LIN {X 0,Y 522.499,Z 557.03,A -85,B 0,C 180,E1 4654.238,E2 4654.238} C_VEL
LIN {X 0,Y 522.631,Z 557.03,A -85,B 0,C 180,E1 4659.658,E2 4659.658} C_VEL
LIN {X 0,Y 522.497,Z 557.03,A -85,B 0,C 180,E1 4664.884,E2 4664.884} C_VEL
LIN {X 0,Y 522.702,Z 557.03,A -85,B 0,C 180,E1 4670.012,E2 4670.012} C_VEL
LIN {X 0,Y 522.868,Z 557.03,A -85,B 0,C 180,E1 4675.016,E2 4675.016} C_VEL
LIN {X 0,Y 522.928,Z 557.03,A -85,B 0,C 180,E1 4680,E2 4680} C_VEL
LIN {X 0,Y 522.866,Z 557.03,A -85,B 0,C 180,E1 4684.983,E2 4684.983} C_VEL
LIN {X 0,Y 522.762,Z 557.03,A -85,B 0,C 180,E1 4690.025,E2 4690.025} C_VEL
LIN {X 0,Y 522.691,Z 557.03,A -85,B 0,C 180,E1 4695.11,E2 4695.11} C_VEL
LIN {X 0,Y 522.622,Z 557.03,A -85,B 0,C 180,E1 4700.341,E2 4700.341} C_VEL
LIN {X 0,Y 522.441,Z 557.03,A -85,B 0,C 180,E1 4706.052,E2 4706.052} C_VEL
LIN {X 0,Y 522.368,Z 557.03,A -85,B 0,C 180,E1 4711.445,E2 4711.445} C_VEL
LIN {X 0,Y 522.262,Z 557.03,A -85,B 0,C 180,E1 4717.499,E2 4717.499} C_VEL
LIN {X 0,Y 522.346,Z 557.03,A -85,B 0,C 180,E1 4723.561,E2 4723.561} C_VEL
LIN {X 0,Y 522.43,Z 557.03,A -85,B 0,C 180,E1 4728.89,E2 4728.89} C_VEL
LIN {X 0,Y 522.316,Z 557.03,A -85,B 0,C 180,E1 4734.567,E2 4734.567} C_VEL
LIN {X 0,Y 522.477,Z 557.132,A -85,B 0,C 180,E1 4740.056,E2 4740.056} C_VEL
LIN {X 0,Y 533.026,Z 584.562,A -85,B 0,C 180,E1 4741.253,E2 4741.253} C_VEL
LIN {X 0,Y 531.972,Z 621.412,A -85,B 0,C 180,E1 4742.156,E2 4742.156} C_VEL
LIN {X 0,Y 530.472,Z 657.437,A -85,B 0,C 180,E1 4743.703,E2 4743.703} C_VEL
LIN {X 0,Y 528.574,Z 691.879,A -85,B 0,C 180,E1 4745.909,E2 4745.909} C_VEL
LIN {X 0,Y 526.76,Z 722.651,A -85,B 0,C 180,E1 4748.647,E2 4748.647} C_VEL
LIN {X 0,Y 525.154,Z 749.674,A -85,B 0,C 180,E1 4751.879,E2 4751.879} C_VEL
LIN {X 0,Y 524.132,Z 770.932,A -85,B 0,C 180,E1 4755.312,E2 4755.312} C_VEL
LIN {X 0,Y 523.51,Z 787.531,A -85,B 0,C 180,E1 4758.998,E2 4758.998} C_VEL
LIN {X 0,Y 523.319,Z 798.445,A -85,B 0,C 180,E1 4762.519,E2 4762.519} C_VEL
LIN {X 0,Y 523.187,Z 805.714,A -85,B 0,C 180,E1 4766.682,E2 4766.682} C_VEL
LIN {X 0,Y 523.118,Z 807.495,A -85,B 0,C 180,E1 4770,E2 4770} C_VEL
LIN {X 0,Y 523.197,Z 804.909,A -85,B 0,C 180,E1 4773.94,E2 4773.94} C_VEL
LIN {X 0,Y 523.423,Z 797.131,A -85,B 0,C 180,E1 4777.897,E2 4777.897} C_VEL
LIN {X 0,Y 523.665,Z 784.536,A -85,B 0,C 180,E1 4781.676,E2 4781.676} C_VEL
LIN {X 0,Y 524.44,Z 765.964,A -85,B 0,C 180,E1 4785.488,E2 4785.488} C_VEL
LIN {X 0,Y 525.654,Z 741.391,A -85,B 0,C 180,E1 4789.125,E2 4789.125} C_VEL
LIN {X 0,Y 527.287,Z 712.977,A -85,B 0,C 180,E1 4792.217,E2 4792.217} C_VEL
LIN {X 0,Y 529.245,Z 680.156,A -85,B 0,C 180,E1 4794.845,E2 4794.845} C_VEL
LIN {X 0,Y 530.944,Z 645.809,A -85,B 0,C 180,E1 4796.786,E2 4796.786} C_VEL
LIN {X 0,Y 532.346,Z 608.713,A -85,B 0,C 180,E1 4798.141,E2 4798.141} C_VEL
LIN {X 0,Y 532.591,Z 581.575,A -85,B 0,C 180,E1 4798.739,E2 4798.739} C_VEL
LIN {X 0,Y 522.511,Z 557.03,A -85,B 0,C 180,E1 4799.925,E2 4799.925} C_VEL
LIN {X 0,Y 522.295,Z 557.03,A -85,B 0,C 180,E1 4805.746,E2 4805.746} C_VEL
LIN {X 0,Y 522.316,Z 557.03,A -85,B 0,C 180,E1 4811.813,E2 4811.813} C_VEL
LIN {X 0,Y 522.415,Z 557.03,A -85,B 0,C 180,E1 4818.2,E2 4818.2} C_VEL
LIN {X 0,Y 522.306,Z 557.03,A -85,B 0,C 180,E1 4824.57,E2 4824.57} C_VEL
LIN {X 0,Y 522.381,Z 557.03,A -85,B 0,C 180,E1 4830.483,E2 4830.483} C_VEL
LIN {X 0,Y 522.584,Z 557.03,A -85,B 0,C 180,E1 4836.073,E2 4836.073} C_VEL
LIN {X 0,Y 522.688,Z 557.03,A -85,B 0,C 180,E1 4841.421,E2 4841.421} C_VEL
LIN {X 0,Y 522.818,Z 557.03,A -85,B 0,C 180,E1 4846.606,E2 4846.606} C_VEL
LIN {X 0,Y 522.822,Z 557.03,A -85,B 0,C 180,E1 4851.675,E2 4851.675} C_VEL
LIN {X 0,Y 523.008,Z 557.03,A -85,B 0,C 180,E1 4856.681,E2 4856.681} C_VEL
LIN {X 0,Y 523.061,Z 557.03,A -85,B 0,C 180,E1 4861.659,E2 4861.659} C_VEL
LIN {X 0,Y 522.914,Z 557.03,A -85,B 0,C 180,E1 4866.651,E2 4866.651} C_VEL
LIN {X 0,Y 522.728,Z 557.03,A -85,B 0,C 180,E1 4871.697,E2 4871.697} C_VEL
LIN {X 0,Y 522.567,Z 557.03,A -85,B 0,C 180,E1 4877.037,E2 4877.037} C_VEL
LIN {X 0,Y 522.584,Z 557.03,A -85,B 0,C 180,E1 4882.124,E2 4882.124} C_VEL
LIN {X 0,Y 522.459,Z 557.03,A -85,B 0,C 180,E1 4887.622,E2 4887.622} C_VEL
LIN {X 0,Y 522.344,Z 557.03,A -85,B 0,C 180,E1 4892.52,E2 4892.52} C_VEL
LIN {X 0,Y 519.879,Z 557.03,A -85,B 0,C 180,E1 4893.934,E2 4893.934} C_VEL
LIN {X 0,Y 514.507,Z 557.03,A -85,B 0,C 180,E1 4896.053,E2 4896.053} C_VEL
LIN {X 0,Y 514.405,Z 557.03,A -85,B 0,C 180,E1 4896.298,E2 4896.298} C_VEL
LIN {X 0,Y 514.489,Z 557.03,A -85,B 0,C 180,E1 4902.634,E2 4902.634} C_VEL
LIN {X 0,Y 514.412,Z 557.03,A -85,B 0,C 180,E1 4907.395,E2 4907.395} C_VEL
LIN {X 0,Y 514.417,Z 557.03,A -85,B 0,C 180,E1 4913.939,E2 4913.939} C_VEL
LIN {X 0,Y 514.455,Z 557.03,A -85,B 0,C 180,E1 4914.47,E2 4914.47} C_VEL
LIN {X 0,Y 527.108,Z 583.904,A -85,B 0,C 180,E1 4915.848,E2 4915.848} C_VEL
LIN {X 0,Y 529.672,Z 589.378,A -85,B 0,C 180,E1 4916.123,E2 4916.123} C_VEL
LIN {X 0,Y 528.629,Z 631.367,A -85,B 0,C 180,E1 4916.994,E2 4916.994} C_VEL
LIN {X 0,Y 526.749,Z 669.423,A -85,B 0,C 180,E1 4918.414,E2 4918.414} C_VEL
LIN {X 0,Y 524.486,Z 706.242,A -85,B 0,C 180,E1 4920.481,E2 4920.481} C_VEL
LIN {X 0,Y 521.855,Z 740.903,A -85,B 0,C 180,E1 4923.16,E2 4923.16} C_VEL
LIN {X 0,Y 519.397,Z 773.263,A -85,B 0,C 180,E1 4926.513,E2 4926.513} C_VEL
LIN {X 0,Y 517.458,Z 800.955,A -85,B 0,C 180,E1 4930.338,E2 4930.338} C_VEL
LIN {X 0,Y 516.251,Z 822.301,A -85,B 0,C 180,E1 4934.26,E2 4934.26} C_VEL
LIN {X 0,Y 515.569,Z 837.902,A -85,B 0,C 180,E1 4938.138,E2 4938.138} C_VEL
LIN {X 0,Y 515.355,Z 849.538,A -85,B 0,C 180,E1 4942.403,E2 4942.403} C_VEL
LIN {X 0,Y 515.273,Z 855.897,A -85,B 0,C 180,E1 4946.631,E2 4946.631} C_VEL
LIN {X 0,Y 515.214,Z 857.5,A -85,B 0,C 180,E1 4950,E2 4950} C_VEL
LIN {X 0,Y 515.205,Z 855.898,A -85,B 0,C 180,E1 4953.37,E2 4953.37} C_VEL
LIN {X 0,Y 515.345,Z 849.538,A -85,B 0,C 180,E1 4957.597,E2 4957.597} C_VEL
LIN {X 0,Y 515.631,Z 837.901,A -85,B 0,C 180,E1 4961.862,E2 4961.862} C_VEL
LIN {X 0,Y 516.397,Z 820.237,A -85,B 0,C 180,E1 4966.173,E2 4966.173} C_VEL
LIN {X 0,Y 517.695,Z 798.153,A -85,B 0,C 180,E1 4970.099,E2 4970.099} C_VEL
LIN {X 0,Y 519.59,Z 771.372,A -85,B 0,C 180,E1 4973.702,E2 4973.702} C_VEL
LIN {X 0,Y 521.839,Z 740.896,A -85,B 0,C 180,E1 4976.842,E2 4976.842} C_VEL
LIN {X 0,Y 524.41,Z 706.227,A -85,B 0,C 180,E1 4979.524,E2 4979.524} C_VEL
LIN {X 0,Y 526.744,Z 669.005,A -85,B 0,C 180,E1 4981.607,E2 4981.607} C_VEL
LIN {X 0,Y 528.668,Z 630.098,A -85,B 0,C 180,E1 4983.042,E2 4983.042} C_VEL
LIN {X 0,Y 529.166,Z 588.175,A -85,B 0,C 180,E1 4983.933,E2 4983.933} C_VEL
LIN {X 0,Y 514.456,Z 557.03,A -85,B 0,C 180,E1 4985.532,E2 4985.532} C_VEL
LIN {X 0,Y 514.375,Z 557.03,A -85,B 0,C 180,E1 4990.359,E2 4990.359} C_VEL
LIN {X 0,Y 514.417,Z 557.03,A -85,B 0,C 180,E1 4995.063,E2 4995.063} C_VEL
LIN {X 0,Y 514.496,Z 557.03,A -85,B 0,C 180,E1 4999.918,E2 4999.918} C_VEL
LIN {X 0,Y 514.385,Z 557.03,A -85,B 0,C 180,E1 5005.998,E2 5005.998} C_VEL
LIN {X 0,Y 514.51,Z 557.03,A -85,B 0,C 180,E1 5011.984,E2 5011.984} C_VEL
LIN {X 0,Y 514.641,Z 557.03,A -85,B 0,C 180,E1 5017.516,E2 5017.516} C_VEL
LIN {X 0,Y 514.742,Z 557.03,A -85,B 0,C 180,E1 5022.895,E2 5022.895} C_VEL
LIN {X 0,Y 514.768,Z 557.03,A -85,B 0,C 180,E1 5029.836,E2 5029.836} C_VEL
LIN {X 0,Y 514.968,Z 557.03,A -85,B 0,C 180,E1 5034.94,E2 5034.94} C_VEL
LIN {X 0,Y 515.032,Z 557.03,A -85,B 0,C 180,E1 5040,E2 5040} C_VEL
LIN {X 0,Y 514.96,Z 557.03,A -85,B 0,C 180,E1 5045.06,E2 5045.06} C_VEL
LIN {X 0,Y 514.869,Z 557.03,A -85,B 0,C 180,E1 5050.161,E2 5050.161} C_VEL
LIN {X 0,Y 514.779,Z 557.03,A -85,B 0,C 180,E1 5055.348,E2 5055.348} C_VEL
LIN {X 0,Y 514.686,Z 557.03,A -85,B 0,C 180,E1 5060.669,E2 5060.669} C_VEL
LIN {X 0,Y 514.537,Z 557.03,A -85,B 0,C 180,E1 5066.19,E2 5066.19} C_VEL
LIN {X 0,Y 514.479,Z 557.03,A -85,B 0,C 180,E1 5071.984,E2 5071.984} C_VEL
LIN {X 0,Y 514.339,Z 557.03,A -85,B 0,C 180,E1 5078.179,E2 5078.179} C_VEL
LIN {X 0,Y 514.408,Z 557.03,A -85,B 0,C 180,E1 5084.937,E2 5084.937} C_VEL
LIN {X 0,Y 514.5,Z 557.03,A -85,B 0,C 180,E1 5089.912,E2 5089.912} C_VEL
LIN {X 0,Y 514.382,Z 557.03,A -85,B 0,C 180,E1 5095.995,E2 5095.995} C_VEL
LIN {X 0,Y 514.531,Z 557.515,A -85,B 0,C 180,E1 5099.458,E2 5099.458} C_VEL
LIN {X 0,Y 526.353,Z 586.45,A -85,B 0,C 180,E1 5100.821,E2 5100.821} C_VEL
LIN {X 0,Y 525.106,Z 622.044,A -85,B 0,C 180,E1 5101.74,E2 5101.74} C_VEL
LIN {X 0,Y 523.259,Z 658.762,A -85,B 0,C 180,E1 5103.386,E2 5103.386} C_VEL
LIN {X 0,Y 521.147,Z 693.261,A -85,B 0,C 180,E1 5105.658,E2 5105.658} C_VEL
LIN {X 0,Y 519.142,Z 724.17,A -85,B 0,C 180,E1 5108.48,E2 5108.48} C_VEL
LIN {X 0,Y 517.4,Z 751.061,A -85,B 0,C 180,E1 5111.804,E2 5111.804} C_VEL
LIN {X 0,Y 516.257,Z 773.247,A -85,B 0,C 180,E1 5115.545,E2 5115.545} C_VEL
LIN {X 0,Y 515.614,Z 789.381,A -85,B 0,C 180,E1 5119.344,E2 5119.344} C_VEL
LIN {X 0,Y 515.396,Z 800.367,A -85,B 0,C 180,E1 5123.252,E2 5123.252} C_VEL
LIN {X 0,Y 515.204,Z 806.579,A -85,B 0,C 180,E1 5127.564,E2 5127.564} C_VEL
LIN {X 0,Y 515.283,Z 806.982,A -85,B 0,C 180,E1 5131.683,E2 5131.683} C_VEL
LIN {X 0,Y 515.352,Z 801.871,A -85,B 0,C 180,E1 5135.902,E2 5135.902} C_VEL
LIN {X 0,Y 515.538,Z 792.198,A -85,B 0,C 180,E1 5139.722,E2 5139.722} C_VEL
LIN {X 0,Y 516.197,Z 775.889,A -85,B 0,C 180,E1 5143.839,E2 5143.839} C_VEL
LIN {X 0,Y 517.179,Z 754.854,A -85,B 0,C 180,E1 5147.543,E2 5147.543} C_VEL
LIN {X 0,Y 518.68,Z 729.937,A -85,B 0,C 180,E1 5150.797,E2 5150.797} C_VEL
LIN {X 0,Y 520.75,Z 699.762,A -85,B 0,C 180,E1 5153.735,E2 5153.735} C_VEL
LIN {X 0,Y 522.778,Z 667.008,A -85,B 0,C 180,E1 5156.05,E2 5156.05} C_VEL
LIN {X 0,Y 524.759,Z 631.374,A -85,B 0,C 180,E1 5157.815,E2 5157.815} C_VEL
LIN {X 0,Y 526.101,Z 597.165,A -85,B 0,C 180,E1 5158.874,E2 5158.874} C_VEL
LIN {X 0,Y 525.587,Z 583.161,A -85,B 0,C 180,E1 5159.205,E2 5159.205} C_VEL
LIN {X 0,Y 514.561,Z 557.03,A -85,B 0,C 180,E1 5160.492,E2 5160.492} C_VEL
LIN {X 0,Y 514.377,Z 557.03,A -85,B 0,C 180,E1 5166.064,E2 5166.064} C_VEL
LIN {X 0,Y 514.409,Z 557.03,A -85,B 0,C 180,E1 5172.628,E2 5172.628} C_VEL
LIN {X 0,Y 514.486,Z 557.03,A -85,B 0,C 180,E1 5177.406,E2 5177.406} C_VEL
LIN {X 0,Y 514.433,Z 557.03,A -85,B 0,C 180,E1 5182.622,E2 5182.622} C_VEL
LIN {X 0,Y 514.431,Z 557.03,A -85,B 0,C 180,E1 5188.595,E2 5188.595} C_VEL
LIN {X 0,Y 514.608,Z 557.03,A -85,B 0,C 180,E1 5193.814,E2 5193.814} C_VEL
LIN {X 0,Y 514.718,Z 557.03,A -85,B 0,C 180,E1 5200.267,E2 5200.267} C_VEL
LIN {X 0,Y 514.888,Z 557.03,A -85,B 0,C 180,E1 5206.395,E2 5206.395} C_VEL
LIN {X 0,Y 514.935,Z 557.03,A -85,B 0,C 180,E1 5211.547,E2 5211.547} C_VEL
LIN {X 0,Y 515.096,Z 557.03,A -85,B 0,C 180,E1 5216.63,E2 5216.63} C_VEL
LIN {X 0,Y 515.079,Z 557.03,A -85,B 0,C 180,E1 5221.971,E2 5221.971} C_VEL
LIN {X 0,Y 515.004,Z 557.03,A -85,B 0,C 180,E1 5226.753,E2 5226.753} C_VEL
LIN {X 0,Y 514.797,Z 557.03,A -85,B 0,C 180,E1 5231.88,E2 5231.88} C_VEL
LIN {X 0,Y 514.671,Z 557.03,A -85,B 0,C 180,E1 5237.107,E2 5237.107} C_VEL
LIN {X 0,Y 514.639,Z 557.03,A -85,B 0,C 180,E1 5242.485,E2 5242.485} C_VEL
LIN {X 0,Y 514.501,Z 557.03,A -85,B 0,C 180,E1 5248.087,E2 5248.087} C_VEL
LIN {X 0,Y 514.384,Z 557.03,A -85,B 0,C 180,E1 5254.002,E2 5254.002} C_VEL
LIN {X 0,Y 514.405,Z 557.03,A -85,B 0,C 180,E1 5256.298,E2 5256.298} C_VEL
LIN {X 0,Y 513.119,Z 557.03,A -85,B 0,C 180,E1 5257.261,E2 5257.261} C_VEL
LIN {X 0,Y 506.5,Z 557.03,A -85,B 0,C 180,E1 5259.885,E2 5259.885} C_VEL
LIN {X 0,Y 506.412,Z 557.03,A -85,B 0,C 180,E1 5260.134,E2 5260.134} C_VEL
LIN {X 0,Y 506.444,Z 557.03,A -85,B 0,C 180,E1 5265.844,E2 5265.844} C_VEL
LIN {X 0,Y 506.405,Z 557.03,A -85,B 0,C 180,E1 5271.108,E2 5271.108} C_VEL
LIN {X 0,Y 506.542,Z 557.03,A -85,B 0,C 180,E1 5273.919,E2 5273.919} C_VEL
LIN {X 0,Y 517.256,Z 579.74,A -85,B 0,C 180,E1 5275.038,E2 5275.038} C_VEL
LIN {X 0,Y 523.116,Z 591.895,A -85,B 0,C 180,E1 5275.681,E2 5275.681} C_VEL
LIN {X 0,Y 521.907,Z 633.932,A -85,B 0,C 180,E1 5276.594,E2 5276.594} C_VEL
LIN {X 0,Y 519.721,Z 673.354,A -85,B 0,C 180,E1 5278.136,E2 5278.136} C_VEL
LIN {X 0,Y 517.139,Z 711.434,A -85,B 0,C 180,E1 5280.392,E2 5280.392} C_VEL
LIN {X 0,Y 514.294,Z 745.785,A -85,B 0,C 180,E1 5283.206,E2 5283.206} C_VEL
LIN {X 0,Y 511.637,Z 776.353,A -85,B 0,C 180,E1 5286.535,E2 5286.535} C_VEL
LIN {X 0,Y 509.707,Z 802.295,A -85,B 0,C 180,E1 5290.252,E2 5290.252} C_VEL
LIN {X 0,Y 508.425,Z 822.302,A -85,B 0,C 180,E1 5294.011,E2 5294.011} C_VEL
LIN {X 0,Y 507.684,Z 839.28,A -85,B 0,C 180,E1 5298.387,E2 5298.387} C_VEL
LIN {X 0,Y 507.455,Z 849.538,A -85,B 0,C 180,E1 5302.284,E2 5302.284} C_VEL
LIN {X 0,Y 507.366,Z 855.897,A -85,B 0,C 180,E1 5306.579,E2 5306.579} C_VEL
LIN {X 0,Y 507.327,Z 857.5,A -85,B 0,C 180,E1 5310,E2 5310} C_VEL
LIN {X 0,Y 507.305,Z 855.898,A -85,B 0,C 180,E1 5313.422,E2 5313.422} C_VEL
LIN {X 0,Y 507.454,Z 849.538,A -85,B 0,C 180,E1 5317.716,E2 5317.716} C_VEL
LIN {X 0,Y 507.781,Z 837.9,A -85,B 0,C 180,E1 5322.048,E2 5322.048} C_VEL
LIN {X 0,Y 508.634,Z 820.236,A -85,B 0,C 180,E1 5326.427,E2 5326.427} C_VEL
LIN {X 0,Y 510.039,Z 798.151,A -85,B 0,C 180,E1 5330.414,E2 5330.414} C_VEL
LIN {X 0,Y 512.212,Z 770.604,A -85,B 0,C 180,E1 5334.158,E2 5334.158} C_VEL
LIN {X 0,Y 514.731,Z 739.628,A -85,B 0,C 180,E1 5337.362,E2 5337.362} C_VEL
LIN {X 0,Y 517.404,Z 706.224,A -85,B 0,C 180,E1 5339.965,E2 5339.965} C_VEL
LIN {X 0,Y 519.9,Z 669.735,A -85,B 0,C 180,E1 5342.035,E2 5342.035} C_VEL
LIN {X 0,Y 521.975,Z 631.3,A -85,B 0,C 180,E1 5343.484,E2 5343.484} C_VEL
LIN {X 0,Y 522.476,Z 590.576,A -85,B 0,C 180,E1 5344.388,E2 5344.388} C_VEL
LIN {X 0,Y 506.611,Z 558.216,A -85,B 0,C 180,E1 5346.039,E2 5346.039} C_VEL
LIN {X 0,Y 506.517,Z 557.03,A -85,B 0,C 180,E1 5346.195,E2 5346.195} C_VEL
LIN {X 0,Y 506.401,Z 557.03,A -85,B 0,C 180,E1 5351.634,E2 5351.634} C_VEL
LIN {X 0,Y 506.522,Z 557.03,A -85,B 0,C 180,E1 5358.356,E2 5358.356} C_VEL
LIN {X 0,Y 506.529,Z 557.03,A -85,B 0,C 180,E1 5363.809,E2 5363.809} C_VEL
LIN {X 0,Y 506.539,Z 557.03,A -85,B 0,C 180,E1 5370.091,E2 5370.091} C_VEL
LIN {X 0,Y 506.665,Z 557.03,A -85,B 0,C 180,E1 5375.271,E2 5375.271} C_VEL
LIN {X 0,Y 506.836,Z 557.03,A -85,B 0,C 180,E1 5380.817,E2 5380.817} C_VEL
LIN {X 0,Y 506.653,Z 557.03,A -85,B 0,C 180,E1 5386.169,E2 5386.169} C_VEL
LIN {X 0,Y 506.871,Z 557.03,A -85,B 0,C 180,E1 5391.411,E2 5391.411} C_VEL
LIN {X 0,Y 507.009,Z 557.03,A -85,B 0,C 180,E1 5396.576,E2 5396.576} C_VEL
LIN {X 0,Y 507.066,Z 557.03,A -85,B 0,C 180,E1 5401.711,E2 5401.711} C_VEL
LIN {X 0,Y 506.963,Z 557.03,A -85,B 0,C 180,E1 5406.86,E2 5406.86} C_VEL
LIN {X 0,Y 506.862,Z 557.03,A -85,B 0,C 180,E1 5412.068,E2 5412.068} C_VEL
LIN {X 0,Y 506.814,Z 557.03,A -85,B 0,C 180,E1 5417.38,E2 5417.38} C_VEL
LIN {X 0,Y 506.721,Z 557.03,A -85,B 0,C 180,E1 5422.855,E2 5422.855} C_VEL
LIN {X 0,Y 506.529,Z 557.03,A -85,B 0,C 180,E1 5428.569,E2 5428.569} C_VEL
LIN {X 0,Y 506.481,Z 557.03,A -85,B 0,C 180,E1 5434.606,E2 5434.606} C_VEL
LIN {X 0,Y 506.383,Z 557.03,A -85,B 0,C 180,E1 5441.127,E2 5441.127} C_VEL
LIN {X 0,Y 506.49,Z 557.03,A -85,B 0,C 180,E1 5446.564,E2 5446.564} C_VEL
LIN {X 0,Y 506.512,Z 557.03,A -85,B 0,C 180,E1 5453.285,E2 5453.285} C_VEL
LIN {X 0,Y 506.577,Z 557.238,A -85,B 0,C 180,E1 5458.831,E2 5458.831} C_VEL
LIN {X 0,Y 519.682,Z 587.9,A -85,B 0,C 180,E1 5460.364,E2 5460.364} C_VEL
LIN {X 0,Y 518.316,Z 625.057,A -85,B 0,C 180,E1 5461.369,E2 5461.369} C_VEL
LIN {X 0,Y 516.256,Z 660.583,A -85,B 0,C 180,E1 5463.033,E2 5463.033} C_VEL
LIN {X 0,Y 513.847,Z 693.357,A -85,B 0,C 180,E1 5465.289,E2 5465.289} C_VEL
LIN {X 0,Y 511.587,Z 724.917,A -85,B 0,C 180,E1 5468.228,E2 5468.228} C_VEL
LIN {X 0,Y 509.742,Z 751.097,A -85,B 0,C 180,E1 5471.527,E2 5471.527} C_VEL
LIN {X 0,Y 508.46,Z 773.243,A -85,B 0,C 180,E1 5475.318,E2 5475.318} C_VEL
LIN {X 0,Y 507.749,Z 789.668,A -85,B 0,C 180,E1 5479.259,E2 5479.259} C_VEL
LIN {X 0,Y 507.5,Z 800.365,A -85,B 0,C 180,E1 5483.146,E2 5483.146} C_VEL
LIN {X 0,Y 507.388,Z 805.711,A -85,B 0,C 180,E1 5486.578,E2 5486.578} C_VEL
LIN {X 0,Y 507.331,Z 807.495,A -85,B 0,C 180,E1 5490,E2 5490} C_VEL
LIN {X 0,Y 507.423,Z 804.612,A -85,B 0,C 180,E1 5494.278,E2 5494.278} C_VEL
LIN {X 0,Y 507.627,Z 795.988,A -85,B 0,C 180,E1 5498.576,E2 5498.576} C_VEL
LIN {X 0,Y 508.021,Z 782.805,A -85,B 0,C 180,E1 5502.478,E2 5502.478} C_VEL
LIN {X 0,Y 508.94,Z 763.523,A -85,B 0,C 180,E1 5506.416,E2 5506.416} C_VEL
LIN {X 0,Y 510.525,Z 739.65,A -85,B 0,C 180,E1 5509.941,E2 5509.941} C_VEL
LIN {X 0,Y 512.532,Z 711.195,A -85,B 0,C 180,E1 5513.072,E2 5513.072} C_VEL
LIN {X 0,Y 515.048,Z 677.433,A -85,B 0,C 180,E1 5515.812,E2 5515.812} C_VEL
LIN {X 0,Y 517.295,Z 643.917,A -85,B 0,C 180,E1 5517.746,E2 5517.746} C_VEL
LIN {X 0,Y 519.049,Z 607.178,A -85,B 0,C 180,E1 5519.113,E2 5519.113} C_VEL
LIN {X 0,Y 519.234,Z 586.102,A -85,B 0,C 180,E1 5519.613,E2 5519.613} C_VEL
LIN {X 0,Y 506.604,Z 557.03,A -85,B 0,C 180,E1 5521.131,E2 5521.131} C_VEL
LIN {X 0,Y 506.454,Z 557.03,A -85,B 0,C 180,E1 5526.719,E2 5526.719} C_VEL
LIN {X 0,Y 506.448,Z 557.03,A -85,B 0,C 180,E1 5533.44,E2 5533.44} C_VEL
LIN {X 0,Y 506.49,Z 557.03,A -85,B 0,C 180,E1 5538.883,E2 5538.883} C_VEL
LIN {X 0,Y 506.463,Z 557.03,A -85,B 0,C 180,E1 5545.392,E2 5545.392} C_VEL
LIN {X 0,Y 506.535,Z 557.03,A -85,B 0,C 180,E1 5551.432,E2 5551.432} C_VEL
LIN {X 0,Y 506.739,Z 557.03,A -85,B 0,C 180,E1 5557.146,E2 5557.146} C_VEL
LIN {X 0,Y 506.886,Z 557.03,A -85,B 0,C 180,E1 5562.906,E2 5562.906} C_VEL
LIN {X 0,Y 506.913,Z 557.03,A -85,B 0,C 180,E1 5567.933,E2 5567.933} C_VEL
LIN {X 0,Y 506.962,Z 557.03,A -85,B 0,C 180,E1 5573.14,E2 5573.14} C_VEL
LIN {X 0,Y 507.06,Z 557.03,A -85,B 0,C 180,E1 5578.289,E2 5578.289} C_VEL
LIN {X 0,Y 507.003,Z 557.03,A -85,B 0,C 180,E1 5583.424,E2 5583.424} C_VEL
LIN {X 0,Y 506.89,Z 557.03,A -85,B 0,C 180,E1 5588.589,E2 5588.589} C_VEL
LIN {X 0,Y 506.826,Z 557.03,A -85,B 0,C 180,E1 5593.826,E2 5593.826} C_VEL
LIN {X 0,Y 506.71,Z 557.03,A -85,B 0,C 180,E1 5599.188,E2 5599.188} C_VEL
LIN {X 0,Y 506.672,Z 557.03,A -85,B 0,C 180,E1 5604.729,E2 5604.729} C_VEL
LIN {X 0,Y 506.529,Z 557.03,A -85,B 0,C 180,E1 5610.538,E2 5610.538} C_VEL
LIN {X 0,Y 506.522,Z 557.03,A -85,B 0,C 180,E1 5616.711,E2 5616.711} C_VEL
LIN {X 0,Y 506.412,Z 557.03,A -85,B 0,C 180,E1 5620.134,E2 5620.134} C_VEL
LIN {X 0,Y 503.923,Z 557.03,A -85,B 0,C 180,E1 5621.594,E2 5621.594} C_VEL
LIN {X 0,Y 498.652,Z 557.03,A -85,B 0,C 180,E1 5623.784,E2 5623.784} C_VEL
LIN {X 0,Y 498.565,Z 557.03,A -85,B 0,C 180,E1 5624.037,E2 5624.037} C_VEL
LIN {X 0,Y 498.446,Z 557.03,A -85,B 0,C 180,E1 5630.366,E2 5630.366} C_VEL
LIN {X 0,Y 498.625,Z 557.617,A -85,B 0,C 180,E1 5633.375,E2 5633.375} C_VEL
LIN {X 0,Y 516.486,Z 594.362,A -85,B 0,C 180,E1 5635.22,E2 5635.22} C_VEL
LIN {X 0,Y 515.178,Z 636.741,A -85,B 0,C 180,E1 5636.191,E2 5636.191} C_VEL
LIN {X 0,Y 512.771,Z 676.295,A -85,B 0,C 180,E1 5637.814,E2 5637.814} C_VEL
LIN {X 0,Y 509.993,Z 712.973,A -85,B 0,C 180,E1 5640.058,E2 5640.058} C_VEL
LIN {X 0,Y 506.953,Z 746.935,A -85,B 0,C 180,E1 5642.906,E2 5642.906} C_VEL
LIN {X 0,Y 504.073,Z 777.662,A -85,B 0,C 180,E1 5646.336,E2 5646.336} C_VEL
LIN {X 0,Y 501.933,Z 804.002,A -85,B 0,C 180,E1 5650.229,E2 5650.229} C_VEL
LIN {X 0,Y 500.594,Z 824.261,A -85,B 0,C 180,E1 5654.205,E2 5654.205} C_VEL
LIN {X 0,Y 499.831,Z 839.281,A -85,B 0,C 180,E1 5658.202,E2 5658.202} C_VEL
LIN {X 0,Y 499.57,Z 849.538,A -85,B 0,C 180,E1 5662.162,E2 5662.162} C_VEL
LIN {X 0,Y 499.459,Z 855.897,A -85,B 0,C 180,E1 5666.524,E2 5666.524} C_VEL
LIN {X 0,Y 499.444,Z 857.5,A -85,B 0,C 180,E1 5670,E2 5670} C_VEL
LIN {X 0,Y 499.405,Z 855.898,A -85,B 0,C 180,E1 5673.477,E2 5673.477} C_VEL
LIN {X 0,Y 499.577,Z 849.538,A -85,B 0,C 180,E1 5677.839,E2 5677.839} C_VEL
LIN {X 0,Y 499.944,Z 837.9,A -85,B 0,C 180,E1 5682.239,E2 5682.239} C_VEL
LIN {X 0,Y 500.898,Z 820.234,A -85,B 0,C 180,E1 5686.688,E2 5686.688} C_VEL
LIN {X 0,Y 502.454,Z 797.834,A -85,B 0,C 180,E1 5690.786,E2 5690.786} C_VEL
LIN {X 0,Y 504.802,Z 770.245,A -85,B 0,C 180,E1 5694.58,E2 5694.58} C_VEL
LIN {X 0,Y 507.55,Z 739.625,A -85,B 0,C 180,E1 5697.782,E2 5697.782} C_VEL
LIN {X 0,Y 510.447,Z 706.323,A -85,B 0,C 180,E1 5700.409,E2 5700.409} C_VEL
LIN {X 0,Y 513.153,Z 669.732,A -85,B 0,C 180,E1 5702.507,E2 5702.507} C_VEL
LIN {X 0,Y 515.405,Z 630.577,A -85,B 0,C 180,E1 5703.991,E2 5703.991} C_VEL
LIN {X 0,Y 515.916,Z 593.113,A -85,B 0,C 180,E1 5704.841,E2 5704.841} C_VEL
LIN {X 0,Y 498.583,Z 557.03,A -85,B 0,C 180,E1 5706.683,E2 5706.683} C_VEL
LIN {X 0,Y 498.512,Z 557.03,A -85,B 0,C 180,E1 5713.208,E2 5713.208} C_VEL
LIN {X 0,Y 498.54,Z 557.03,A -85,B 0,C 180,E1 5719.398,E2 5719.398} C_VEL
LIN {X 0,Y 498.587,Z 557.03,A -85,B 0,C 180,E1 5725.076,E2 5725.076} C_VEL
LIN {X 0,Y 498.612,Z 557.03,A -85,B 0,C 180,E1 5731.715,E2 5731.715} C_VEL
LIN {X 0,Y 498.762,Z 557.03,A -85,B 0,C 180,E1 5736.758,E2 5736.758} C_VEL
LIN {X 0,Y 498.889,Z 557.03,A -85,B 0,C 180,E1 5742.334,E2 5742.334} C_VEL
LIN {X 0,Y 498.798,Z 557.03,A -85,B 0,C 180,E1 5747.733,E2 5747.733} C_VEL
LIN {X 0,Y 499.15,Z 557.03,A -85,B 0,C 180,E1 5753.031,E2 5753.031} C_VEL
LIN {X 0,Y 499.404,Z 557.03,A -85,B 0,C 180,E1 5758.262,E2 5758.262} C_VEL
LIN {X 0,Y 499.3,Z 557.03,A -85,B 0,C 180,E1 5763.476,E2 5763.476} C_VEL
LIN {X 0,Y 499.096,Z 557.03,A -85,B 0,C 180,E1 5768.723,E2 5768.723} C_VEL
LIN {X 0,Y 498.969,Z 557.03,A -85,B 0,C 180,E1 5774.047,E2 5774.047} C_VEL
LIN {X 0,Y 498.835,Z 557.03,A -85,B 0,C 180,E1 5779.795,E2 5779.795} C_VEL
LIN {X 0,Y 498.727,Z 557.03,A -85,B 0,C 180,E1 5785.149,E2 5785.149} C_VEL
LIN {X 0,Y 498.566,Z 557.03,A -85,B 0,C 180,E1 5791.754,E2 5791.754} C_VEL
LIN {X 0,Y 498.448,Z 557.03,A -85,B 0,C 180,E1 5797.837,E2 5797.837} C_VEL
LIN {X 0,Y 498.524,Z 557.03,A -85,B 0,C 180,E1 5804.304,E2 5804.304} C_VEL
LIN {X 0,Y 498.531,Z 557.03,A -85,B 0,C 180,E1 5810.373,E2 5810.373} C_VEL
LIN {X 0,Y 498.566,Z 557.03,A -85,B 0,C 180,E1 5816.864,E2 5816.864} C_VEL
LIN {X 0,Y 498.65,Z 557.03,A -85,B 0,C 180,E1 5818.152,E2 5818.152} C_VEL
LIN {X 0,Y 512.972,Z 589.835,A -85,B 0,C 180,E1 5819.894,E2 5819.894} C_VEL
LIN {X 0,Y 511.545,Z 628.105,A -85,B 0,C 180,E1 5820.993,E2 5820.993} C_VEL
LIN {X 0,Y 509.316,Z 662.339,A -85,B 0,C 180,E1 5822.659,E2 5822.659} C_VEL
LIN {X 0,Y 506.728,Z 694.383,A -85,B 0,C 180,E1 5824.918,E2 5824.918} C_VEL
LIN {X 0,Y 504.116,Z 725.151,A -85,B 0,C 180,E1 5827.914,E2 5827.914} C_VEL
LIN {X 0,Y 501.992,Z 752.226,A -85,B 0,C 180,E1 5831.408,E2 5831.408} C_VEL
LIN {X 0,Y 500.726,Z 772.632,A -85,B 0,C 180,E1 5834.961,E2 5834.961} C_VEL
LIN {X 0,Y 499.913,Z 788.129,A -85,B 0,C 180,E1 5838.646,E2 5838.646} C_VEL
LIN {X 0,Y 499.663,Z 798.439,A -85,B 0,C 180,E1 5842.163,E2 5842.163} C_VEL
LIN {X 0,Y 499.499,Z 805.71,A -85,B 0,C 180,E1 5846.524,E2 5846.524} C_VEL
LIN {X 0,Y 499.442,Z 807.495,A -85,B 0,C 180,E1 5850,E2 5850} C_VEL
LIN {X 0,Y 499.542,Z 804.613,A -85,B 0,C 180,E1 5854.345,E2 5854.345} C_VEL
LIN {X 0,Y 499.749,Z 795.99,A -85,B 0,C 180,E1 5858.712,E2 5858.712} C_VEL
LIN {X 0,Y 500.182,Z 782.808,A -85,B 0,C 180,E1 5862.677,E2 5862.677} C_VEL
LIN {X 0,Y 501.213,Z 763.526,A -85,B 0,C 180,E1 5866.677,E2 5866.677} C_VEL
LIN {X 0,Y 502.923,Z 739.656,A -85,B 0,C 180,E1 5870.255,E2 5870.255} C_VEL
LIN {X 0,Y 505.531,Z 708.354,A -85,B 0,C 180,E1 5873.754,E2 5873.754} C_VEL
LIN {X 0,Y 508.176,Z 677.074,A -85,B 0,C 180,E1 5876.307,E2 5876.307} C_VEL
LIN {X 0,Y 510.644,Z 643.292,A -85,B 0,C 180,E1 5878.259,E2 5878.259} C_VEL
LIN {X 0,Y 512.475,Z 607.469,A -85,B 0,C 180,E1 5879.598,E2 5879.598} C_VEL
LIN {X 0,Y 512.746,Z 588.544,A -85,B 0,C 180,E1 5880.058,E2 5880.058} C_VEL
LIN {X 0,Y 498.704,Z 557.03,A -85,B 0,C 180,E1 5881.788,E2 5881.788} C_VEL
LIN {X 0,Y 498.449,Z 557.03,A -85,B 0,C 180,E1 5887.843,E2 5887.843} C_VEL
LIN {X 0,Y 498.551,Z 557.03,A -85,B 0,C 180,E1 5894.305,E2 5894.305} C_VEL
LIN {X 0,Y 498.524,Z 557.03,A -85,B 0,C 180,E1 5900.377,E2 5900.377} C_VEL
LIN {X 0,Y 498.525,Z 557.03,A -85,B 0,C 180,E1 5906.864,E2 5906.864} C_VEL
LIN {X 0,Y 498.665,Z 557.03,A -85,B 0,C 180,E1 5912.91,E2 5912.91} C_VEL
LIN {X 0,Y 498.865,Z 557.03,A -85,B 0,C 180,E1 5918.644,E2 5918.644} C_VEL
LIN {X 0,Y 498.99,Z 557.03,A -85,B 0,C 180,E1 5924.154,E2 5924.154} C_VEL
LIN {X 0,Y 499.067,Z 557.03,A -85,B 0,C 180,E1 5929.513,E2 5929.513} C_VEL
LIN {X 0,Y 499.149,Z 557.03,A -85,B 0,C 180,E1 5934.78,E2 5934.78} C_VEL
LIN {X 0,Y 499.277,Z 557.03,A -85,B 0,C 180,E1 5940,E2 5940} C_VEL
LIN {X 0,Y 499.166,Z 557.03,A -85,B 0,C 180,E1 5945.221,E2 5945.221} C_VEL
LIN {X 0,Y 499.013,Z 557.03,A -85,B 0,C 180,E1 5950.488,E2 5950.488} C_VEL
LIN {X 0,Y 498.87,Z 557.03,A -85,B 0,C 180,E1 5955.851,E2 5955.851} C_VEL
LIN {X 0,Y 498.799,Z 557.03,A -85,B 0,C 180,E1 5961.36,E2 5961.36} C_VEL
LIN {X 0,Y 498.652,Z 557.03,A -85,B 0,C 180,E1 5967.092,E2 5967.092} C_VEL
LIN {X 0,Y 498.538,Z 557.03,A -85,B 0,C 180,E1 5973.136,E2 5973.136} C_VEL
LIN {X 0,Y 498.537,Z 557.03,A -85,B 0,C 180,E1 5979.623,E2 5979.623} C_VEL
LIN {X 0,Y 498.565,Z 557.03,A -85,B 0,C 180,E1 5984.037,E2 5984.037} C_VEL
LIN {X 0,Y 496.1,Z 557.03,A -85,B 0,C 180,E1 5985.511,E2 5985.511} C_VEL
LIN {X 0,Y 490.589,Z 557.03,A -85,B 0,C 180,E1 5987.977,E2 5987.977} C_VEL
LIN {X 0,Y 490.617,Z 557.03,A -85,B 0,C 180,E1 5992.765,E2 5992.765} C_VEL
LIN {X 0,Y 509.78,Z 598.268,A -85,B 0,C 180,E1 5994.835,E2 5994.835} C_VEL
LIN {X 0,Y 508.329,Z 638.786,A -85,B 0,C 180,E1 5995.79,E2 5995.79} C_VEL
LIN {X 0,Y 506.046,Z 675.877,A -85,B 0,C 180,E1 5997.309,E2 5997.309} C_VEL
LIN {X 0,Y 503.027,Z 712.969,A -85,B 0,C 180,E1 5999.6,E2 5999.6} C_VEL
LIN {X 0,Y 499.691,Z 747.167,A -85,B 0,C 180,E1 6002.504,E2 6002.504} C_VEL
LIN {X 0,Y 496.638,Z 777.704,A -85,B 0,C 180,E1 6005.966,E2 6005.966} C_VEL
LIN {X 0,Y 494.276,Z 804.226,A -85,B 0,C 180,E1 6009.95,E2 6009.95} C_VEL
LIN {X 0,Y 492.797,Z 824.26,A -85,B 0,C 180,E1 6013.948,E2 6013.948} C_VEL
LIN {X 0,Y 491.971,Z 839.281,A -85,B 0,C 180,E1 6018.011,E2 6018.011} C_VEL
LIN {X 0,Y 491.678,Z 849.538,A -85,B 0,C 180,E1 6022.035,E2 6022.035} C_VEL
LIN {X 0,Y 491.553,Z 855.897,A -85,B 0,C 180,E1 6026.469,E2 6026.469} C_VEL
LIN {X 0,Y 491.544,Z 857.5,A -85,B 0,C 180,E1 6030,E2 6030} C_VEL
LIN {X 0,Y 491.504,Z 855.899,A -85,B 0,C 180,E1 6033.532,E2 6033.532} C_VEL
LIN {X 0,Y 491.69,Z 849.538,A -85,B 0,C 180,E1 6037.965,E2 6037.965} C_VEL
LIN {X 0,Y 492.113,Z 837.899,A -85,B 0,C 180,E1 6042.437,E2 6042.437} C_VEL
LIN {X 0,Y 493.132,Z 820.233,A -85,B 0,C 180,E1 6046.959,E2 6046.959} C_VEL
LIN {X 0,Y 494.845,Z 797.833,A -85,B 0,C 180,E1 6051.121,E2 6051.121} C_VEL
LIN {X 0,Y 497.296,Z 771.445,A -85,B 0,C 180,E1 6054.826,E2 6054.826} C_VEL
LIN {X 0,Y 500.342,Z 740.256,A -85,B 0,C 180,E1 6058.156,E2 6058.156} C_VEL
LIN {X 0,Y 503.53,Z 706.32,A -85,B 0,C 180,E1 6060.872,E2 6060.872} C_VEL
LIN {X 0,Y 506.456,Z 669.495,A -85,B 0,C 180,E1 6063.004,E2 6063.004} C_VEL
LIN {X 0,Y 508.642,Z 631.11,A -85,B 0,C 180,E1 6064.442,E2 6064.442} C_VEL
LIN {X 0,Y 509.102,Z 595.771,A -85,B 0,C 180,E1 6065.254,E2 6065.254} C_VEL
LIN {X 0,Y 490.609,Z 557.03,A -85,B 0,C 180,E1 6067.287,E2 6067.287} C_VEL
LIN {X 0,Y 490.571,Z 557.03,A -85,B 0,C 180,E1 6072.765,E2 6072.765} C_VEL
LIN {X 0,Y 490.691,Z 557.03,A -85,B 0,C 180,E1 6077.777,E2 6077.777} C_VEL
LIN {X 0,Y 490.593,Z 557.03,A -85,B 0,C 180,E1 6084.103,E2 6084.103} C_VEL
LIN {X 0,Y 490.633,Z 557.03,A -85,B 0,C 180,E1 6090.415,E2 6090.415} C_VEL
LIN {X 0,Y 490.834,Z 557.03,A -85,B 0,C 180,E1 6096.36,E2 6096.36} C_VEL
LIN {X 0,Y 490.972,Z 557.03,A -85,B 0,C 180,E1 6102.039,E2 6102.039} C_VEL
LIN {X 0,Y 490.888,Z 557.03,A -85,B 0,C 180,E1 6107.532,E2 6107.532} C_VEL
LIN {X 0,Y 491.223,Z 557.03,A -85,B 0,C 180,E1 6112.918,E2 6112.918} C_VEL
LIN {X 0,Y 491.492,Z 557.03,A -85,B 0,C 180,E1 6118.235,E2 6118.235} C_VEL
LIN {X 0,Y 491.387,Z 557.03,A -85,B 0,C 180,E1 6123.532,E2 6123.532} C_VEL
LIN {X 0,Y 491.113,Z 557.03,A -85,B 0,C 180,E1 6129.414,E2 6129.414} C_VEL
LIN {X 0,Y 491.036,Z 557.03,A -85,B 0,C 180,E1 6134.279,E2 6134.279} C_VEL
LIN {X 0,Y 490.931,Z 557.03,A -85,B 0,C 180,E1 6139.829,E2 6139.829} C_VEL
LIN {X 0,Y 490.755,Z 557.03,A -85,B 0,C 180,E1 6145.587,E2 6145.587} C_VEL
LIN {X 0,Y 490.687,Z 557.03,A -85,B 0,C 180,E1 6151.635,E2 6151.635} C_VEL
LIN {X 0,Y 490.518,Z 557.03,A -85,B 0,C 180,E1 6158.118,E2 6158.118} C_VEL
LIN {X 0,Y 490.614,Z 557.03,A -85,B 0,C 180,E1 6164.782,E2 6164.782} C_VEL
LIN {X 0,Y 490.617,Z 557.03,A -85,B 0,C 180,E1 6170.484,E2 6170.484} C_VEL
LIN {X 0,Y 490.619,Z 557.03,A -85,B 0,C 180,E1 6176.424,E2 6176.424} C_VEL
LIN {X 0,Y 490.732,Z 557.79,A -85,B 0,C 180,E1 6177.518,E2 6177.518} C_VEL
LIN {X 0,Y 506.489,Z 592.242,A -85,B 0,C 180,E1 6179.435,E2 6179.435} C_VEL
LIN {X 0,Y 504.86,Z 629.676,A -85,B 0,C 180,E1 6180.551,E2 6180.551} C_VEL
LIN {X 0,Y 502.435,Z 664.21,A -85,B 0,C 180,E1 6182.277,E2 6182.277} C_VEL
LIN {X 0,Y 499.641,Z 695.659,A -85,B 0,C 180,E1 6184.553,E2 6184.553} C_VEL
LIN {X 0,Y 496.783,Z 726.33,A -85,B 0,C 180,E1 6187.606,E2 6187.606} C_VEL
LIN {X 0,Y 494.276,Z 753.025,A -85,B 0,C 180,E1 6191.232,E2 6191.232} C_VEL
LIN {X 0,Y 492.835,Z 774.861,A -85,B 0,C 180,E1 6195.182,E2 6195.182} C_VEL
LIN {X 0,Y 491.962,Z 791.132,A -85,B 0,C 180,E1 6199.359,E2 6199.359} C_VEL
LIN {X 0,Y 491.71,Z 800.363,A -85,B 0,C 180,E1 6202.925,E2 6202.925} C_VEL
LIN {X 0,Y 491.597,Z 805.709,A -85,B 0,C 180,E1 6206.468,E2 6206.468} C_VEL
LIN {X 0,Y 491.542,Z 807.495,A -85,B 0,C 180,E1 6210,E2 6210} C_VEL
LIN {X 0,Y 491.661,Z 804.613,A -85,B 0,C 180,E1 6214.415,E2 6214.415} C_VEL
LIN {X 0,Y 491.859,Z 795.992,A -85,B 0,C 180,E1 6218.853,E2 6218.853} C_VEL
LIN {X 0,Y 492.364,Z 782.81,A -85,B 0,C 180,E1 6222.882,E2 6222.882} C_VEL
LIN {X 0,Y 493.493,Z 763.53,A -85,B 0,C 180,E1 6226.945,E2 6226.945} C_VEL
LIN {X 0,Y 495.64,Z 737.212,A -85,B 0,C 180,E1 6230.954,E2 6230.954} C_VEL
LIN {X 0,Y 498.43,Z 708.155,A -85,B 0,C 180,E1 6234.235,E2 6234.235} C_VEL
LIN {X 0,Y 501.341,Z 677.056,A -85,B 0,C 180,E1 6236.795,E2 6236.795} C_VEL
LIN {X 0,Y 503.941,Z 643.978,A -85,B 0,C 180,E1 6238.731,E2 6238.731} C_VEL
LIN {X 0,Y 505.935,Z 607.777,A -85,B 0,C 180,E1 6240.098,E2 6240.098} C_VEL
LIN {X 0,Y 505.968,Z 590.288,A -85,B 0,C 180,E1 6240.555,E2 6240.555} C_VEL
LIN {X 0,Y 490.724,Z 557.03,A -85,B 0,C 180,E1 6242.415,E2 6242.415} C_VEL
LIN {X 0,Y 490.521,Z 557.03,A -85,B 0,C 180,E1 6248.121,E2 6248.121} C_VEL
LIN {X 0,Y 490.63,Z 557.03,A -85,B 0,C 180,E1 6252.758,E2 6252.758} C_VEL
LIN {X 0,Y 490.682,Z 557.03,A -85,B 0,C 180,E1 6257.777,E2 6257.777} C_VEL
LIN {X 0,Y 490.563,Z 557.03,A -85,B 0,C 180,E1 6264.101,E2 6264.101} C_VEL
LIN {X 0,Y 490.627,Z 557.03,A -85,B 0,C 180,E1 6270.415,E2 6270.415} C_VEL
LIN {X 0,Y 490.857,Z 557.03,A -85,B 0,C 180,E1 6276.362,E2 6276.362} C_VEL
LIN {X 0,Y 491.007,Z 557.03,A -85,B 0,C 180,E1 6282.041,E2 6282.041} C_VEL
LIN {X 0,Y 491.091,Z 557.03,A -85,B 0,C 180,E1 6287.538,E2 6287.538} C_VEL
LIN {X 0,Y 491.143,Z 557.03,A -85,B 0,C 180,E1 6292.918,E2 6292.918} C_VEL
LIN {X 0,Y 491.273,Z 557.03,A -85,B 0,C 180,E1 6298.234,E2 6298.234} C_VEL
LIN {X 0,Y 491.203,Z 557.03,A -85,B 0,C 180,E1 6303.534,E2 6303.534} C_VEL
LIN {X 0,Y 491.05,Z 557.03,A -85,B 0,C 180,E1 6309.374,E2 6309.374} C_VEL
LIN {X 0,Y 490.974,Z 557.03,A -85,B 0,C 180,E1 6314.282,E2 6314.282} C_VEL
LIN {X 0,Y 490.863,Z 557.03,A -85,B 0,C 180,E1 6319.833,E2 6319.833} C_VEL
LIN {X 0,Y 490.777,Z 557.03,A -85,B 0,C 180,E1 6325.587,E2 6325.587} C_VEL
LIN {X 0,Y 490.661,Z 557.03,A -85,B 0,C 180,E1 6331.638,E2 6331.638} C_VEL
LIN {X 0,Y 490.603,Z 557.03,A -85,B 0,C 180,E1 6338.111,E2 6338.111} C_VEL
LIN {X 0,Y 490.588,Z 557.03,A -85,B 0,C 180,E1 6344.039,E2 6344.039} C_VEL
LIN {X 0,Y 490.589,Z 557.03,A -85,B 0,C 180,E1 6347.977,E2 6347.977} C_VEL
LIN {X 0,Y 486.498,Z 557.03,A -85,B 0,C 180,E1 6349.957,E2 6349.957} C_VEL
LIN {X 0,Y 482.646,Z 557.03,A -85,B 0,C 180,E1 6351.969,E2 6351.969} C_VEL
LIN {X 0,Y 482.693,Z 557.604,A -85,B 0,C 180,E1 6352.175,E2 6352.175} C_VEL
LIN {X 0,Y 502.955,Z 600.842,A -85,B 0,C 180,E1 6354.419,E2 6354.419} C_VEL
LIN {X 0,Y 501.345,Z 640.778,A -85,B 0,C 180,E1 6355.412,E2 6355.412} C_VEL
LIN {X 0,Y 498.869,Z 678.75,A -85,B 0,C 180,E1 6357.017,E2 6357.017} C_VEL
LIN {X 0,Y 496.083,Z 712.966,A -85,B 0,C 180,E1 6359.129,E2 6359.129} C_VEL
LIN {X 0,Y 492.687,Z 745.776,A -85,B 0,C 180,E1 6361.929,E2 6361.929} C_VEL
LIN {X 0,Y 489.481,Z 775.737,A -85,B 0,C 180,E1 6365.319,E2 6365.319} C_VEL
LIN {X 0,Y 486.87,Z 801.77,A -85,B 0,C 180,E1 6369.191,E2 6369.191} C_VEL
LIN {X 0,Y 485.193,Z 822.305,A -85,B 0,C 180,E1 6373.223,E2 6373.223} C_VEL
LIN {X 0,Y 484.118,Z 839.281,A -85,B 0,C 180,E1 6377.813,E2 6377.813} C_VEL
LIN {X 0,Y 483.803,Z 849.538,A -85,B 0,C 180,E1 6381.905,E2 6381.905} C_VEL
LIN {X 0,Y 483.646,Z 855.897,A -85,B 0,C 180,E1 6386.411,E2 6386.411} C_VEL
LIN {X 0,Y 483.661,Z 857.5,A -85,B 0,C 180,E1 6390,E2 6390} C_VEL
LIN {X 0,Y 483.609,Z 855.899,A -85,B 0,C 180,E1 6393.59,E2 6393.59} C_VEL
LIN {X 0,Y 483.818,Z 849.538,A -85,B 0,C 180,E1 6398.096,E2 6398.096} C_VEL
LIN {X 0,Y 484.286,Z 837.899,A -85,B 0,C 180,E1 6402.642,E2 6402.642} C_VEL
LIN {X 0,Y 485.356,Z 820.264,A -85,B 0,C 180,E1 6407.232,E2 6407.232} C_VEL
LIN {X 0,Y 487.255,Z 797.904,A -85,B 0,C 180,E1 6411.454,E2 6411.454} C_VEL
LIN {X 0,Y 489.974,Z 771.08,A -85,B 0,C 180,E1 6415.269,E2 6415.269} C_VEL
LIN {X 0,Y 493.303,Z 739.595,A -85,B 0,C 180,E1 6418.66,E2 6418.66} C_VEL
LIN {X 0,Y 496.629,Z 706.181,A -85,B 0,C 180,E1 6421.357,E2 6421.357} C_VEL
LIN {X 0,Y 499.522,Z 668.996,A -85,B 0,C 180,E1 6423.464,E2 6423.464} C_VEL
LIN {X 0,Y 501.855,Z 629.758,A -85,B 0,C 180,E1 6424.932,E2 6424.932} C_VEL
LIN {X 0,Y 502.329,Z 598.28,A -85,B 0,C 180,E1 6425.675,E2 6425.675} C_VEL
LIN {X 0,Y 482.656,Z 557.03,A -85,B 0,C 180,E1 6427.932,E2 6427.932} C_VEL
LIN {X 0,Y 482.621,Z 557.03,A -85,B 0,C 180,E1 6433.822,E2 6433.822} C_VEL
LIN {X 0,Y 482.704,Z 557.03,A -85,B 0,C 180,E1 6438.833,E2 6438.833} C_VEL
LIN {X 0,Y 482.635,Z 557.03,A -85,B 0,C 180,E1 6444.651,E2 6444.651} C_VEL
LIN {X 0,Y 482.722,Z 557.03,A -85,B 0,C 180,E1 6449.88,E2 6449.88} C_VEL
LIN {X 0,Y 482.873,Z 557.03,A -85,B 0,C 180,E1 6455.946,E2 6455.946} C_VEL
LIN {X 0,Y 483.034,Z 557.03,A -85,B 0,C 180,E1 6461.734,E2 6461.734} C_VEL
LIN {X 0,Y 482.956,Z 557.03,A -85,B 0,C 180,E1 6467.324,E2 6467.324} C_VEL
LIN {X 0,Y 483.304,Z 557.03,A -85,B 0,C 180,E1 6472.802,E2 6472.802} C_VEL
LIN {X 0,Y 483.583,Z 557.03,A -85,B 0,C 180,E1 6478.206,E2 6478.206} C_VEL
LIN {X 0,Y 483.499,Z 557.03,A -85,B 0,C 180,E1 6483.59,E2 6483.59} C_VEL
LIN {X 0,Y 483.253,Z 557.03,A -85,B 0,C 180,E1 6489.012,E2 6489.012} C_VEL
LIN {X 0,Y 483.108,Z 557.03,A -85,B 0,C 180,E1 6494.519,E2 6494.519} C_VEL
LIN {X 0,Y 482.993,Z 557.03,A -85,B 0,C 180,E1 6500.169,E2 6500.169} C_VEL
LIN {X 0,Y 482.841,Z 557.03,A -85,B 0,C 180,E1 6506.038,E2 6506.038} C_VEL
LIN {X 0,Y 482.722,Z 557.03,A -85,B 0,C 180,E1 6512.219,E2 6512.219} C_VEL
LIN {X 0,Y 482.591,Z 557.03,A -85,B 0,C 180,E1 6518.86,E2 6518.86} C_VEL
LIN {X 0,Y 482.618,Z 557.03,A -85,B 0,C 180,E1 6523.817,E2 6523.817} C_VEL
LIN {X 0,Y 482.712,Z 557.03,A -85,B 0,C 180,E1 6528.826,E2 6528.826} C_VEL
LIN {X 0,Y 482.629,Z 557.03,A -85,B 0,C 180,E1 6534.645,E2 6534.645} C_VEL
LIN {X 0,Y 482.747,Z 557.03,A -85,B 0,C 180,E1 6536.803,E2 6536.803} C_VEL
LIN {X 0,Y 489.551,Z 571.514,A -85,B 0,C 180,E1 6537.647,E2 6537.647} C_VEL
LIN {X 0,Y 499.882,Z 594.315,A -85,B 0,C 180,E1 6538.945,E2 6538.945} C_VEL
LIN {X 0,Y 498.268,Z 630.672,A -85,B 0,C 180,E1 6540.07,E2 6540.07} C_VEL
LIN {X 0,Y 495.701,Z 664.364,A -85,B 0,C 180,E1 6541.774,E2 6541.774} C_VEL
LIN {X 0,Y 492.625,Z 696.698,A -85,B 0,C 180,E1 6544.148,E2 6544.148} C_VEL
LIN {X 0,Y 489.486,Z 727.22,A -85,B 0,C 180,E1 6547.254,E2 6547.254} C_VEL
LIN {X 0,Y 486.746,Z 753.675,A -85,B 0,C 180,E1 6550.937,E2 6550.937} C_VEL
LIN {X 0,Y 484.982,Z 775.913,A -85,B 0,C 180,E1 6555.163,E2 6555.163} C_VEL
LIN {X 0,Y 484.097,Z 791.13,A -85,B 0,C 180,E1 6559.184,E2 6559.184} C_VEL
LIN {X 0,Y 483.823,Z 800.361,A -85,B 0,C 180,E1 6562.809,E2 6562.809} C_VEL
LIN {X 0,Y 483.715,Z 805.708,A -85,B 0,C 180,E1 6566.411,E2 6566.411} C_VEL
LIN {X 0,Y 483.658,Z 807.494,A -85,B 0,C 180,E1 6570,E2 6570} C_VEL
LIN {X 0,Y 483.776,Z 804.614,A -85,B 0,C 180,E1 6574.487,E2 6574.487} C_VEL
LIN {X 0,Y 483.985,Z 795.994,A -85,B 0,C 180,E1 6578.999,E2 6578.999} C_VEL
LIN {X 0,Y 484.547,Z 782.812,A -85,B 0,C 180,E1 6583.093,E2 6583.093} C_VEL
LIN {X 0,Y 485.943,Z 762.523,A -85,B 0,C 180,E1 6587.45,E2 6587.45} C_VEL
LIN {X 0,Y 488.202,Z 738.589,A -85,B 0,C 180,E1 6591.211,E2 6591.211} C_VEL
LIN {X 0,Y 491.314,Z 709.267,A -85,B 0,C 180,E1 6594.609,E2 6594.609} C_VEL
LIN {X 0,Y 494.482,Z 677.88,A -85,B 0,C 180,E1 6597.243,E2 6597.243} C_VEL
LIN {X 0,Y 497.315,Z 644.248,A -85,B 0,C 180,E1 6599.237,E2 6599.237} C_VEL
LIN {X 0,Y 499.413,Z 608.763,A -85,B 0,C 180,E1 6600.594,E2 6600.594} C_VEL
LIN {X 0,Y 499.494,Z 592.538,A -85,B 0,C 180,E1 6601.037,E2 6601.037} C_VEL
LIN {X 0,Y 482.93,Z 558.596,A -85,B 0,C 180,E1 6603.044,E2 6603.044} C_VEL
LIN {X 0,Y 482.77,Z 557.03,A -85,B 0,C 180,E1 6603.093,E2 6603.093} C_VEL
LIN {X 0,Y 482.596,Z 557.03,A -85,B 0,C 180,E1 6608.863,E2 6608.863} C_VEL
LIN {X 0,Y 482.656,Z 557.03,A -85,B 0,C 180,E1 6613.827,E2 6613.827} C_VEL
LIN {X 0,Y 482.712,Z 557.03,A -85,B 0,C 180,E1 6618.831,E2 6618.831} C_VEL
LIN {X 0,Y 482.609,Z 557.03,A -85,B 0,C 180,E1 6624.654,E2 6624.654} C_VEL
LIN {X 0,Y 482.711,Z 557.03,A -85,B 0,C 180,E1 6629.88,E2 6629.88} C_VEL
LIN {X 0,Y 482.896,Z 557.03,A -85,B 0,C 180,E1 6635.948,E2 6635.948} C_VEL
LIN {X 0,Y 483.069,Z 557.03,A -85,B 0,C 180,E1 6641.736,E2 6641.736} C_VEL
LIN {X 0,Y 483.17,Z 557.03,A -85,B 0,C 180,E1 6647.33,E2 6647.33} C_VEL
LIN {X 0,Y 483.244,Z 557.03,A -85,B 0,C 180,E1 6652.801,E2 6652.801} C_VEL
LIN {X 0,Y 483.387,Z 557.03,A -85,B 0,C 180,E1 6658.206,E2 6658.206} C_VEL
LIN {X 0,Y 483.308,Z 557.03,A -85,B 0,C 180,E1 6663.592,E2 6663.592} C_VEL
LIN {X 0,Y 483.175,Z 557.03,A -85,B 0,C 180,E1 6669.014,E2 6669.014} C_VEL
LIN {X 0,Y 483.055,Z 557.03,A -85,B 0,C 180,E1 6674.521,E2 6674.521} C_VEL
LIN {X 0,Y 482.947,Z 557.03,A -85,B 0,C 180,E1 6680.172,E2 6680.172} C_VEL
LIN {X 0,Y 482.862,Z 557.03,A -85,B 0,C 180,E1 6686.037,E2 6686.037} C_VEL
LIN {X 0,Y 482.707,Z 557.03,A -85,B 0,C 180,E1 6692.221,E2 6692.221} C_VEL
LIN {X 0,Y 482.678,Z 557.03,A -85,B 0,C 180,E1 6698.852,E2 6698.852} C_VEL
LIN {X 0,Y 482.689,Z 557.03,A -85,B 0,C 180,E1 6703.827,E2 6703.827} C_VEL
LIN {X 0,Y 482.615,Z 557.03,A -85,B 0,C 180,E1 6708.84,E2 6708.84} C_VEL
LIN {X 0,Y 482.646,Z 557.03,A -85,B 0,C 180,E1 6711.969,E2 6711.969} C_VEL
LIN {X 0,Y 484.845,Z 559.912,A -85,B 0,C 180,E1 6712.385,E2 6712.385} C_VEL
LIN {X 0,Y 487.245,Z 569.61,A -85,B 0,C 180,E1 6712.738,E2 6712.738} C_VEL
LIN {X 0,Y 488.946,Z 587.257,A -85,B 0,C 180,E1 6713.166,E2 6713.166} C_VEL
LIN {X 0,Y 489.802,Z 589.484,A -85,B 0,C 180,E1 6713.272,E2 6713.272} C_VEL
LIN {X 0,Y 496.144,Z 602.104,A -85,B 0,C 180,E1 6713.964,E2 6713.964} C_VEL
LIN {X 0,Y 494.358,Z 642.495,A -85,B 0,C 180,E1 6715.011,E2 6715.011} C_VEL
LIN {X 0,Y 491.726,Z 680.428,A -85,B 0,C 180,E1 6716.673,E2 6716.673} C_VEL
LIN {X 0,Y 488.544,Z 717.049,A -85,B 0,C 180,E1 6719.009,E2 6719.009} C_VEL
LIN {X 0,Y 485.507,Z 746.225,A -85,B 0,C 180,E1 6721.526,E2 6721.526} C_VEL
LIN {X 0,Y 482.11,Z 775.743,A -85,B 0,C 180,E1 6724.916,E2 6724.916} C_VEL
LIN {X 0,Y 479.262,Z 802.007,A -85,B 0,C 180,E1 6728.888,E2 6728.888} C_VEL
LIN {X 0,Y 477.436,Z 822.638,A -85,B 0,C 180,E1 6733.023,E2 6733.023} C_VEL
LIN {X 0,Y 476.261,Z 839.282,A -85,B 0,C 180,E1 6737.609,E2 6737.609} C_VEL
LIN {X 0,Y 475.932,Z 849.538,A -85,B 0,C 180,E1 6741.77,E2 6741.77} C_VEL
LIN {X 0,Y 475.74,Z 855.898,A -85,B 0,C 180,E1 6746.351,E2 6746.351} C_VEL
LIN {X 0,Y 475.761,Z 857.5,A -85,B 0,C 180,E1 6750,E2 6750} C_VEL
LIN {X 0,Y 475.707,Z 855.899,A -85,B 0,C 180,E1 6753.65,E2 6753.65} C_VEL
LIN {X 0,Y 475.948,Z 849.539,A -85,B 0,C 180,E1 6758.231,E2 6758.231} C_VEL
LIN {X 0,Y 476.462,Z 837.898,A -85,B 0,C 180,E1 6762.853,E2 6762.853} C_VEL
LIN {X 0,Y 477.582,Z 821.039,A -85,B 0,C 180,E1 6767.351,E2 6767.351} C_VEL
LIN {X 0,Y 479.686,Z 797.9,A -85,B 0,C 180,E1 6771.811,E2 6771.811} C_VEL
LIN {X 0,Y 482.731,Z 770.335,A -85,B 0,C 180,E1 6775.772,E2 6775.772} C_VEL
LIN {X 0,Y 486.309,Z 738.898,A -85,B 0,C 180,E1 6779.181,E2 6779.181} C_VEL
LIN {X 0,Y 489.592,Z 705.359,A -85,B 0,C 180,E1 6781.824,E2 6781.824} C_VEL
LIN {X 0,Y 492.583,Z 668.74,A -85,B 0,C 180,E1 6783.917,E2 6783.917} C_VEL
LIN {X 0,Y 495.097,Z 628.568,A -85,B 0,C 180,E1 6785.43,E2 6785.43} C_VEL
LIN {X 0,Y 495.643,Z 600.928,A -85,B 0,C 180,E1 6786.096,E2 6786.096} C_VEL
LIN {X 0,Y 474.727,Z 557.03,A -85,B 0,C 180,E1 6788.541,E2 6788.541} C_VEL
LIN {X 0,Y 474.676,Z 557.03,A -85,B 0,C 180,E1 6795.438,E2 6795.438} C_VEL
LIN {X 0,Y 474.7,Z 557.03,A -85,B 0,C 180,E1 6800.368,E2 6800.368} C_VEL
LIN {X 0,Y 474.7,Z 557.03,A -85,B 0,C 180,E1 6806.024,E2 6806.024} C_VEL
LIN {X 0,Y 474.802,Z 557.03,A -85,B 0,C 180,E1 6811.426,E2 6811.426} C_VEL
LIN {X 0,Y 475.017,Z 557.03,A -85,B 0,C 180,E1 6817.569,E2 6817.569} C_VEL
LIN {X 0,Y 475.066,Z 557.03,A -85,B 0,C 180,E1 6823.332,E2 6823.332} C_VEL
LIN {X 0,Y 475.152,Z 557.03,A -85,B 0,C 180,E1 6828.978,E2 6828.978} C_VEL
LIN {X 0,Y 475.444,Z 557.03,A -85,B 0,C 180,E1 6834.518,E2 6834.518} C_VEL
LIN {X 0,Y 475.585,Z 557.03,A -85,B 0,C 180,E1 6840,E2 6840} C_VEL
LIN {X 0,Y 475.417,Z 557.03,A -85,B 0,C 180,E1 6845.482,E2 6845.482} C_VEL
LIN {X 0,Y 475.24,Z 557.03,A -85,B 0,C 180,E1 6851.019,E2 6851.019} C_VEL
LIN {X 0,Y 475.103,Z 557.03,A -85,B 0,C 180,E1 6857.052,E2 6857.052} C_VEL
LIN {X 0,Y 475.013,Z 557.03,A -85,B 0,C 180,E1 6862.486,E2 6862.486} C_VEL
LIN {X 0,Y 474.797,Z 557.03,A -85,B 0,C 180,E1 6868.573,E2 6868.573} C_VEL
LIN {X 0,Y 474.711,Z 557.03,A -85,B 0,C 180,E1 6875.033,E2 6875.033} C_VEL
LIN {X 0,Y 474.59,Z 557.03,A -85,B 0,C 180,E1 6882.059,E2 6882.059} C_VEL
LIN {X 0,Y 474.695,Z 557.03,A -85,B 0,C 180,E1 6887.948,E2 6887.948} C_VEL
LIN {X 0,Y 474.716,Z 557.03,A -85,B 0,C 180,E1 6894.964,E2 6894.964} C_VEL
LIN {X 0,Y 474.801,Z 557.03,A -85,B 0,C 180,E1 6896.114,E2 6896.114} C_VEL
LIN {X 0,Y 480.784,Z 570.121,A -85,B 0,C 180,E1 6896.873,E2 6896.873} C_VEL
LIN {X 0,Y 493.435,Z 596.699,A -85,B 0,C 180,E1 6898.466,E2 6898.466} C_VEL
LIN {X 0,Y 491.62,Z 633.13,A -85,B 0,C 180,E1 6899.635,E2 6899.635} C_VEL
LIN {X 0,Y 488.963,Z 665.54,A -85,B 0,C 180,E1 6901.317,E2 6901.317} C_VEL
LIN {X 0,Y 485.553,Z 698.424,A -85,B 0,C 180,E1 6903.789,E2 6903.789} C_VEL
LIN {X 0,Y 482.226,Z 728.183,A -85,B 0,C 180,E1 6906.892,E2 6906.892} C_VEL
LIN {X 0,Y 479.258,Z 754.413,A -85,B 0,C 180,E1 6910.627,E2 6910.627} C_VEL
LIN {X 0,Y 477.284,Z 775.99,A -85,B 0,C 180,E1 6914.828,E2 6914.828} C_VEL
LIN {X 0,Y 476.203,Z 792.314,A -85,B 0,C 180,E1 6919.408,E2 6919.408} C_VEL
LIN {X 0,Y 475.926,Z 802.027,A -85,B 0,C 180,E1 6923.607,E2 6923.607} C_VEL
LIN {X 0,Y 475.769,Z 807.034,A -85,B 0,C 180,E1 6928.176,E2 6928.176} C_VEL
LIN {X 0,Y 475.812,Z 806.981,A -85,B 0,C 180,E1 6931.823,E2 6931.823} C_VEL
LIN {X 0,Y 475.909,Z 801.875,A -85,B 0,C 180,E1 6936.393,E2 6936.393} C_VEL
LIN {X 0,Y 476.231,Z 791.958,A -85,B 0,C 180,E1 6940.624,E2 6940.624} C_VEL
LIN {X 0,Y 477.371,Z 775.586,A -85,B 0,C 180,E1 6945.168,E2 6945.168} C_VEL
LIN {X 0,Y 479.217,Z 755.291,A -85,B 0,C 180,E1 6949.134,E2 6949.134} C_VEL
LIN {X 0,Y 481.807,Z 731.205,A -85,B 0,C 180,E1 6952.64,E2 6952.64} C_VEL
LIN {X 0,Y 485.069,Z 702.605,A -85,B 0,C 180,E1 6955.743,E2 6955.743} C_VEL
LIN {X 0,Y 488.558,Z 669.74,A -85,B 0,C 180,E1 6958.329,E2 6958.329} C_VEL
LIN {X 0,Y 491.519,Z 635.502,A -85,B 0,C 180,E1 6960.169,E2 6960.169} C_VEL
LIN {X 0,Y 493.391,Z 601.434,A -85,B 0,C 180,E1 6961.319,E2 6961.319} C_VEL
LIN {X 0,Y 492.943,Z 594.682,A -85,B 0,C 180,E1 6961.54,E2 6961.54} C_VEL
LIN {X 0,Y 474.816,Z 557.03,A -85,B 0,C 180,E1 6963.815,E2 6963.815} C_VEL
LIN {X 0,Y 474.607,Z 557.03,A -85,B 0,C 180,E1 6970.043,E2 6970.043} C_VEL
LIN {X 0,Y 474.689,Z 557.03,A -85,B 0,C 180,E1 6975.441,E2 6975.441} C_VEL
LIN {X 0,Y 474.694,Z 557.03,A -85,B 0,C 180,E1 6980.368,E2 6980.368} C_VEL
LIN {X 0,Y 474.703,Z 557.03,A -85,B 0,C 180,E1 6987.169,E2 6987.169} C_VEL
LIN {X 0,Y 474.89,Z 557.03,A -85,B 0,C 180,E1 6993.493,E2 6993.493} C_VEL
LIN {X 0,Y 475.105,Z 557.03,A -85,B 0,C 180,E1 6999.481,E2 6999.481} C_VEL
LIN {X 0,Y 475.266,Z 557.03,A -85,B 0,C 180,E1 7005.236,E2 7005.236} C_VEL
LIN {X 0,Y 475.334,Z 557.03,A -85,B 0,C 180,E1 7011.237,E2 7011.237} C_VEL
LIN {X 0,Y 475.581,Z 557.03,A -85,B 0,C 180,E1 7016.35,E2 7016.35} C_VEL
LIN {X 0,Y 475.666,Z 557.03,A -85,B 0,C 180,E1 7021.824,E2 7021.824} C_VEL
LIN {X 0,Y 475.383,Z 557.03,A -85,B 0,C 180,E1 7027.319,E2 7027.319} C_VEL
LIN {X 0,Y 475.171,Z 557.03,A -85,B 0,C 180,E1 7032.887,E2 7032.887} C_VEL
LIN {X 0,Y 475.033,Z 557.03,A -85,B 0,C 180,E1 7038.585,E2 7038.585} C_VEL
LIN {X 0,Y 474.975,Z 557.03,A -85,B 0,C 180,E1 7044.48,E2 7044.48} C_VEL
LIN {X 0,Y 474.774,Z 557.03,A -85,B 0,C 180,E1 7050.678,E2 7050.678} C_VEL
LIN {X 0,Y 474.734,Z 557.03,A -85,B 0,C 180,E1 7057.295,E2 7057.295} C_VEL
LIN {X 0,Y 474.7,Z 557.03,A -85,B 0,C 180,E1 7062.813,E2 7062.813} C_VEL
LIN {X 0,Y 474.634,Z 557.03,A -85,B 0,C 180,E1 7067.942,E2 7067.942} C_VEL
LIN {X 0,Y 474.719,Z 557.03,A -85,B 0,C 180,E1 7071.509,E2 7071.509} C_VEL
LIN {X 0,Y 489.802,Z 589.484,A -85,B 0,C 180,E1 7073.272,E2 7073.272} C_VEL
LIN {X 0,Y 491.086,Z 597.817,A -85,B 0,C 180,E1 7073.513,E2 7073.513} C_VEL
LIN {X 0,Y 489.119,Z 612.892,A -85,B 0,C 180,E1 7073.699,E2 7073.699} C_VEL
LIN {X 0,Y 486.966,Z 651.744,A -85,B 0,C 180,E1 7074.887,E2 7074.887} C_VEL
LIN {X 0,Y 483.84,Z 690.458,A -85,B 0,C 180,E1 7076.797,E2 7076.797} C_VEL
LIN {X 0,Y 480.312,Z 726.658,A -85,B 0,C 180,E1 7079.361,E2 7079.361} C_VEL
LIN {X 0,Y 476.705,Z 759.572,A -85,B 0,C 180,E1 7082.517,E2 7082.517} C_VEL
LIN {X 0,Y 473.407,Z 786.643,A -85,B 0,C 180,E1 7086.041,E2 7086.041} C_VEL
LIN {X 0,Y 470.751,Z 811.201,A -85,B 0,C 180,E1 7090.263,E2 7090.263} C_VEL
LIN {X 0,Y 469.15,Z 829.832,A -85,B 0,C 180,E1 7094.559,E2 7094.559} C_VEL
LIN {X 0,Y 468.272,Z 843.215,A -85,B 0,C 180,E1 7098.814,E2 7098.814} C_VEL
LIN {X 0,Y 467.938,Z 852.721,A -85,B 0,C 180,E1 7103.498,E2 7103.498} C_VEL
LIN {X 0,Y 467.868,Z 857.086,A -85,B 0,C 180,E1 7108.146,E2 7108.146} C_VEL
LIN {X 0,Y 467.912,Z 857.086,A -85,B 0,C 180,E1 7111.855,E2 7111.855} C_VEL
LIN {X 0,Y 467.95,Z 852.724,A -85,B 0,C 180,E1 7116.503,E2 7116.503} C_VEL
LIN {X 0,Y 468.267,Z 843.213,A -85,B 0,C 180,E1 7121.187,E2 7121.187} C_VEL
LIN {X 0,Y 469.262,Z 828.091,A -85,B 0,C 180,E1 7125.918,E2 7125.918} C_VEL
LIN {X 0,Y 471.257,Z 806.261,A -85,B 0,C 180,E1 7130.696,E2 7130.696} C_VEL
LIN {X 0,Y 474.151,Z 780.987,A -85,B 0,C 180,E1 7134.778,E2 7134.778} C_VEL
LIN {X 0,Y 477.462,Z 752.889,A -85,B 0,C 180,E1 7138.207,E2 7138.207} C_VEL
LIN {X 0,Y 481.099,Z 718.708,A -85,B 0,C 180,E1 7141.279,E2 7141.279} C_VEL
LIN {X 0,Y 484.587,Z 682.09,A -85,B 0,C 180,E1 7143.682,E2 7143.682} C_VEL
LIN {X 0,Y 487.523,Z 643.123,A -85,B 0,C 180,E1 7145.433,E2 7145.433} C_VEL
LIN {X 0,Y 488.944,Z 603.674,A -85,B 0,C 180,E1 7146.524,E2 7146.524} C_VEL
LIN {X 0,Y 466.748,Z 557.03,A -85,B 0,C 180,E1 7149.193,E2 7149.193} C_VEL
LIN {X 0,Y 466.766,Z 557.03,A -85,B 0,C 180,E1 7155.53,E2 7155.53} C_VEL
LIN {X 0,Y 466.739,Z 557.03,A -85,B 0,C 180,E1 7161.953,E2 7161.953} C_VEL
LIN {X 0,Y 466.797,Z 557.03,A -85,B 0,C 180,E1 7168.74,E2 7168.74} C_VEL
LIN {X 0,Y 467.014,Z 557.03,A -85,B 0,C 180,E1 7175.198,E2 7175.198} C_VEL
LIN {X 0,Y 467.16,Z 557.03,A -85,B 0,C 180,E1 7181.09,E2 7181.09} C_VEL
LIN {X 0,Y 467.106,Z 557.03,A -85,B 0,C 180,E1 7186.886,E2 7186.886} C_VEL
LIN {X 0,Y 467.453,Z 557.03,A -85,B 0,C 180,E1 7192.556,E2 7192.556} C_VEL
LIN {X 0,Y 467.77,Z 557.03,A -85,B 0,C 180,E1 7198.145,E2 7198.145} C_VEL
LIN {X 0,Y 467.699,Z 557.03,A -85,B 0,C 180,E1 7203.712,E2 7203.712} C_VEL
LIN {X 0,Y 467.408,Z 557.03,A -85,B 0,C 180,E1 7209.32,E2 7209.32} C_VEL
LIN {X 0,Y 467.237,Z 557.03,A -85,B 0,C 180,E1 7215.023,E2 7215.023} C_VEL
LIN {X 0,Y 467.113,Z 557.03,A -85,B 0,C 180,E1 7220.886,E2 7220.886} C_VEL
LIN {X 0,Y 466.925,Z 557.03,A -85,B 0,C 180,E1 7226.996,E2 7226.996} C_VEL
LIN {X 0,Y 466.8,Z 557.03,A -85,B 0,C 180,E1 7233.459,E2 7233.459} C_VEL
LIN {X 0,Y 466.653,Z 557.03,A -85,B 0,C 180,E1 7240.455,E2 7240.455} C_VEL
LIN {X 0,Y 466.802,Z 557.03,A -85,B 0,C 180,E1 7247.068,E2 7247.068} C_VEL
LIN {X 0,Y 466.732,Z 557.03,A -85,B 0,C 180,E1 7251.95,E2 7251.95} C_VEL
LIN {X 0,Y 466.85,Z 557.232,A -85,B 0,C 180,E1 7255.399,E2 7255.399} C_VEL
LIN {X 0,Y 473.441,Z 571.166,A -85,B 0,C 180,E1 7256.244,E2 7256.244} C_VEL
LIN {X 0,Y 487.042,Z 599.254,A -85,B 0,C 180,E1 7257.989,E2 7257.989} C_VEL
LIN {X 0,Y 485.015,Z 635.303,A -85,B 0,C 180,E1 7259.177,E2 7259.177} C_VEL
LIN {X 0,Y 482.059,Z 669.024,A -85,B 0,C 180,E1 7260.996,E2 7260.996} C_VEL
LIN {X 0,Y 478.326,Z 701.889,A -85,B 0,C 180,E1 7263.572,E2 7263.572} C_VEL
LIN {X 0,Y 474.743,Z 730.978,A -85,B 0,C 180,E1 7266.755,E2 7266.755} C_VEL
LIN {X 0,Y 471.786,Z 755.198,A -85,B 0,C 180,E1 7270.308,E2 7270.308} C_VEL
LIN {X 0,Y 469.608,Z 776.61,A -85,B 0,C 180,E1 7274.574,E2 7274.574} C_VEL
LIN {X 0,Y 468.46,Z 791.614,A -85,B 0,C 180,E1 7278.818,E2 7278.818} C_VEL
LIN {X 0,Y 468.052,Z 802.133,A -85,B 0,C 180,E1 7283.499,E2 7283.499} C_VEL
LIN {X 0,Y 467.883,Z 807.033,A -85,B 0,C 180,E1 7288.145,E2 7288.145} C_VEL
LIN {X 0,Y 467.919,Z 807.007,A -85,B 0,C 180,E1 7291.854,E2 7291.854} C_VEL
LIN {X 0,Y 468.041,Z 801.99,A -85,B 0,C 180,E1 7296.501,E2 7296.501} C_VEL
LIN {X 0,Y 468.505,Z 791.368,A -85,B 0,C 180,E1 7301.18,E2 7301.18} C_VEL
LIN {X 0,Y 469.811,Z 775.166,A -85,B 0,C 180,E1 7305.658,E2 7305.658} C_VEL
LIN {X 0,Y 471.898,Z 754.689,A -85,B 0,C 180,E1 7309.687,E2 7309.687} C_VEL
LIN {X 0,Y 475.044,Z 728.479,A -85,B 0,C 180,E1 7313.478,E2 7313.478} C_VEL
LIN {X 0,Y 478.73,Z 698.313,A -85,B 0,C 180,E1 7316.66,E2 7316.66} C_VEL
LIN {X 0,Y 482.284,Z 665.946,A -85,B 0,C 180,E1 7319.116,E2 7319.116} C_VEL
LIN {X 0,Y 485.386,Z 631.552,A -85,B 0,C 180,E1 7320.883,E2 7320.883} C_VEL
LIN {X 0,Y 486.642,Z 597.611,A -85,B 0,C 180,E1 7321.999,E2 7321.999} C_VEL
LIN {X 0,Y 466.945,Z 558.244,A -85,B 0,C 180,E1 7324.481,E2 7324.481} C_VEL
LIN {X 0,Y 466.856,Z 557.03,A -85,B 0,C 180,E1 7324.559,E2 7324.559} C_VEL
LIN {X 0,Y 466.678,Z 557.03,A -85,B 0,C 180,E1 7330.456,E2 7330.456} C_VEL
LIN {X 0,Y 466.806,Z 557.03,A -85,B 0,C 180,E1 7337.073,E2 7337.073} C_VEL
LIN {X 0,Y 466.726,Z 557.03,A -85,B 0,C 180,E1 7341.953,E2 7341.953} C_VEL
LIN {X 0,Y 466.785,Z 557.03,A -85,B 0,C 180,E1 7348.74,E2 7348.74} C_VEL
LIN {X 0,Y 467.053,Z 557.03,A -85,B 0,C 180,E1 7355.186,E2 7355.186} C_VEL
LIN {X 0,Y 467.196,Z 557.03,A -85,B 0,C 180,E1 7361.092,E2 7361.092} C_VEL
LIN {X 0,Y 467.336,Z 557.03,A -85,B 0,C 180,E1 7366.894,E2 7366.894} C_VEL
LIN {X 0,Y 467.421,Z 557.03,A -85,B 0,C 180,E1 7372.556,E2 7372.556} C_VEL
LIN {X 0,Y 467.615,Z 557.03,A -85,B 0,C 180,E1 7378.145,E2 7378.145} C_VEL
LIN {X 0,Y 467.496,Z 557.03,A -85,B 0,C 180,E1 7383.714,E2 7383.714} C_VEL
LIN {X 0,Y 467.342,Z 557.03,A -85,B 0,C 180,E1 7389.322,E2 7389.322} C_VEL
LIN {X 0,Y 467.187,Z 557.03,A -85,B 0,C 180,E1 7395.026,E2 7395.026} C_VEL
LIN {X 0,Y 467.082,Z 557.03,A -85,B 0,C 180,E1 7400.888,E2 7400.888} C_VEL
LIN {X 0,Y 466.939,Z 557.03,A -85,B 0,C 180,E1 7406.996,E2 7406.996} C_VEL
LIN {X 0,Y 466.784,Z 557.03,A -85,B 0,C 180,E1 7413.461,E2 7413.461} C_VEL
LIN {X 0,Y 466.759,Z 557.03,A -85,B 0,C 180,E1 7420.444,E2 7420.444} C_VEL
LIN {X 0,Y 466.766,Z 557.03,A -85,B 0,C 180,E1 7427.065,E2 7427.065} C_VEL
LIN {X 0,Y 466.763,Z 557.03,A -85,B 0,C 180,E1 7430.807,E2 7430.807} C_VEL
LIN {X 0,Y 489.339,Z 606.037,A -85,B 0,C 180,E1 7433.553,E2 7433.553} C_VEL
LIN {X 0,Y 489.119,Z 612.892,A -85,B 0,C 180,E1 7433.699,E2 7433.699} C_VEL
LIN {X 0,Y 484.78,Z 629.82,A -85,B 0,C 180,E1 7433.887,E2 7433.887} C_VEL
LIN {X 0,Y 480.648,Z 644.447,A -85,B 0,C 180,E1 7434.141,E2 7434.141} C_VEL
LIN {X 0,Y 480.435,Z 646.55,A -85,B 0,C 180,E1 7434.21,E2 7434.21} C_VEL
LIN {X 0,Y 477.076,Z 687.623,A -85,B 0,C 180,E1 7436.174,E2 7436.174} C_VEL
LIN {X 0,Y 473.3,Z 724.698,A -85,B 0,C 180,E1 7438.787,E2 7438.787} C_VEL
LIN {X 0,Y 469.517,Z 757.456,A -85,B 0,C 180,E1 7441.924,E2 7441.924} C_VEL
LIN {X 0,Y 465.968,Z 786.441,A -85,B 0,C 180,E1 7445.603,E2 7445.603} C_VEL
LIN {X 0,Y 463.09,Z 811.199,A -85,B 0,C 180,E1 7449.923,E2 7449.923} C_VEL
LIN {X 0,Y 461.337,Z 829.831,A -85,B 0,C 180,E1 7454.291,E2 7454.291} C_VEL
LIN {X 0,Y 460.376,Z 844.363,A -85,B 0,C 180,E1 7459.1,E2 7459.1} C_VEL
LIN {X 0,Y 460.041,Z 852.72,A -85,B 0,C 180,E1 7463.386,E2 7463.386} C_VEL
LIN {X 0,Y 459.963,Z 857.086,A -85,B 0,C 180,E1 7468.114,E2 7468.114} C_VEL
LIN {X 0,Y 460.006,Z 857.086,A -85,B 0,C 180,E1 7471.887,E2 7471.887} C_VEL
LIN {X 0,Y 460.05,Z 852.724,A -85,B 0,C 180,E1 7476.615,E2 7476.615} C_VEL
LIN {X 0,Y 460.435,Z 843.213,A -85,B 0,C 180,E1 7481.379,E2 7481.379} C_VEL
LIN {X 0,Y 461.515,Z 828.092,A -85,B 0,C 180,E1 7486.192,E2 7486.192} C_VEL
LIN {X 0,Y 463.665,Z 806.26,A -85,B 0,C 180,E1 7491.051,E2 7491.051} C_VEL
LIN {X 0,Y 466.735,Z 780.825,A -85,B 0,C 180,E1 7495.199,E2 7495.199} C_VEL
LIN {X 0,Y 470.345,Z 750.008,A -85,B 0,C 180,E1 7498.872,E2 7498.872} C_VEL
LIN {X 0,Y 474.183,Z 716.239,A -85,B 0,C 180,E1 7501.887,E2 7501.887} C_VEL
LIN {X 0,Y 477.752,Z 680.323,A -85,B 0,C 180,E1 7504.233,E2 7504.233} C_VEL
LIN {X 0,Y 480.813,Z 641.57,A -85,B 0,C 180,E1 7505.962,E2 7505.962} C_VEL
LIN {X 0,Y 482.038,Z 606.011,A -85,B 0,C 180,E1 7506.987,E2 7506.987} C_VEL
LIN {X 0,Y 458.788,Z 557.03,A -85,B 0,C 180,E1 7509.964,E2 7509.964} C_VEL
LIN {X 0,Y 458.864,Z 557.03,A -85,B 0,C 180,E1 7516.545,E2 7516.545} C_VEL
LIN {X 0,Y 458.807,Z 557.03,A -85,B 0,C 180,E1 7522.373,E2 7522.373} C_VEL
LIN {X 0,Y 458.875,Z 557.03,A -85,B 0,C 180,E1 7529.079,E2 7529.079} C_VEL
LIN {X 0,Y 459.053,Z 557.03,A -85,B 0,C 180,E1 7534.612,E2 7534.612} C_VEL
LIN {X 0,Y 459.252,Z 557.03,A -85,B 0,C 180,E1 7540.752,E2 7540.752} C_VEL
LIN {X 0,Y 459.195,Z 557.03,A -85,B 0,C 180,E1 7546.656,E2 7546.656} C_VEL
LIN {X 0,Y 459.525,Z 557.03,A -85,B 0,C 180,E1 7552.427,E2 7552.427} C_VEL
LIN {X 0,Y 459.858,Z 557.03,A -85,B 0,C 180,E1 7558.113,E2 7558.113} C_VEL
LIN {X 0,Y 459.782,Z 557.03,A -85,B 0,C 180,E1 7563.776,E2 7563.776} C_VEL
LIN {X 0,Y 459.505,Z 557.03,A -85,B 0,C 180,E1 7569.482,E2 7569.482} C_VEL
LIN {X 0,Y 459.304,Z 557.03,A -85,B 0,C 180,E1 7575.289,E2 7575.289} C_VEL
LIN {X 0,Y 459.158,Z 557.03,A -85,B 0,C 180,E1 7581.265,E2 7581.265} C_VEL
LIN {X 0,Y 458.976,Z 557.03,A -85,B 0,C 180,E1 7587.503,E2 7587.503} C_VEL
LIN {X 0,Y 458.804,Z 557.03,A -85,B 0,C 180,E1 7594.122,E2 7594.122} C_VEL
LIN {X 0,Y 458.74,Z 557.03,A -85,B 0,C 180,E1 7600.614,E2 7600.614} C_VEL
LIN {X 0,Y 458.857,Z 557.03,A -85,B 0,C 180,E1 7606.54,E2 7606.54} C_VEL
LIN {X 0,Y 458.799,Z 557.03,A -85,B 0,C 180,E1 7612.368,E2 7612.368} C_VEL
LIN {X 0,Y 458.868,Z 557.146,A -85,B 0,C 180,E1 7614.638,E2 7614.638} C_VEL
LIN {X 0,Y 463.653,Z 567.371,A -85,B 0,C 180,E1 7615.279,E2 7615.279} C_VEL
LIN {X 0,Y 480.349,Z 601.131,A -85,B 0,C 180,E1 7617.469,E2 7617.469} C_VEL
LIN {X 0,Y 478.233,Z 638.966,A -85,B 0,C 180,E1 7618.784,E2 7618.784} C_VEL
LIN {X 0,Y 474.899,Z 674.026,A -85,B 0,C 180,E1 7620.778,E2 7620.778} C_VEL
LIN {X 0,Y 471.2,Z 704.312,A -85,B 0,C 180,E1 7623.266,E2 7623.266} C_VEL
LIN {X 0,Y 467.499,Z 731.994,A -85,B 0,C 180,E1 7626.373,E2 7626.373} C_VEL
LIN {X 0,Y 464.135,Z 757.397,A -85,B 0,C 180,E1 7630.218,E2 7630.218} C_VEL
LIN {X 0,Y 461.924,Z 777.264,A -85,B 0,C 180,E1 7634.311,E2 7634.311} C_VEL
LIN {X 0,Y 460.647,Z 792.147,A -85,B 0,C 180,E1 7638.626,E2 7638.626} C_VEL
LIN {X 0,Y 460.205,Z 802.605,A -85,B 0,C 180,E1 7643.387,E2 7643.387} C_VEL
LIN {X 0,Y 459.992,Z 807.433,A -85,B 0,C 180,E1 7648.113,E2 7648.113} C_VEL
LIN {X 0,Y 460.025,Z 807.382,A -85,B 0,C 180,E1 7651.886,E2 7651.886} C_VEL
LIN {X 0,Y 460.198,Z 802.467,A -85,B 0,C 180,E1 7656.612,E2 7656.612} C_VEL
LIN {X 0,Y 460.7,Z 791.904,A -85,B 0,C 180,E1 7661.372,E2 7661.372} C_VEL
LIN {X 0,Y 462.131,Z 775.842,A -85,B 0,C 180,E1 7665.925,E2 7665.925} C_VEL
LIN {X 0,Y 464.419,Z 755.493,A -85,B 0,C 180,E1 7670.017,E2 7670.017} C_VEL
LIN {X 0,Y 467.58,Z 731.358,A -85,B 0,C 180,E1 7673.622,E2 7673.622} C_VEL
LIN {X 0,Y 471.583,Z 701.425,A -85,B 0,C 180,E1 7676.925,E2 7676.925} C_VEL
LIN {X 0,Y 475.344,Z 669.319,A -85,B 0,C 180,E1 7679.453,E2 7679.453} C_VEL
LIN {X 0,Y 478.498,Z 636.483,A -85,B 0,C 180,E1 7681.224,E2 7681.224} C_VEL
LIN {X 0,Y 480.127,Z 600.032,A -85,B 0,C 180,E1 7682.489,E2 7682.489} C_VEL
LIN {X 0,Y 458.944,Z 557.992,A -85,B 0,C 180,E1 7685.245,E2 7685.245} C_VEL
LIN {X 0,Y 458.86,Z 557.03,A -85,B 0,C 180,E1 7685.494,E2 7685.494} C_VEL
LIN {X 0,Y 458.791,Z 557.03,A -85,B 0,C 180,E1 7691.301,E2 7691.301} C_VEL
LIN {X 0,Y 458.865,Z 557.03,A -85,B 0,C 180,E1 7696.544,E2 7696.544} C_VEL
LIN {X 0,Y 458.792,Z 557.03,A -85,B 0,C 180,E1 7702.374,E2 7702.374} C_VEL
LIN {X 0,Y 458.864,Z 557.03,A -85,B 0,C 180,E1 7709.079,E2 7709.079} C_VEL
LIN {X 0,Y 459.062,Z 557.03,A -85,B 0,C 180,E1 7714.614,E2 7714.614} C_VEL
LIN {X 0,Y 459.288,Z 557.03,A -85,B 0,C 180,E1 7720.754,E2 7720.754} C_VEL
LIN {X 0,Y 459.438,Z 557.03,A -85,B 0,C 180,E1 7726.664,E2 7726.664} C_VEL
LIN {X 0,Y 459.507,Z 557.03,A -85,B 0,C 180,E1 7732.427,E2 7732.427} C_VEL
LIN {X 0,Y 459.713,Z 557.03,A -85,B 0,C 180,E1 7738.113,E2 7738.113} C_VEL
LIN {X 0,Y 459.589,Z 557.03,A -85,B 0,C 180,E1 7743.778,E2 7743.778} C_VEL
LIN {X 0,Y 459.419,Z 557.03,A -85,B 0,C 180,E1 7749.484,E2 7749.484} C_VEL
LIN {X 0,Y 459.249,Z 557.03,A -85,B 0,C 180,E1 7755.292,E2 7755.292} C_VEL
LIN {X 0,Y 459.133,Z 557.03,A -85,B 0,C 180,E1 7761.267,E2 7761.267} C_VEL
LIN {X 0,Y 458.987,Z 557.03,A -85,B 0,C 180,E1 7767.503,E2 7767.503} C_VEL
LIN {X 0,Y 458.802,Z 557.03,A -85,B 0,C 180,E1 7774.123,E2 7774.123} C_VEL
LIN {X 0,Y 458.875,Z 557.03,A -85,B 0,C 180,E1 7780.635,E2 7780.635} C_VEL
LIN {X 0,Y 458.84,Z 557.03,A -85,B 0,C 180,E1 7786.543,E2 7786.543} C_VEL
LIN {X 0,Y 458.826,Z 557.03,A -85,B 0,C 180,E1 7790.076,E2 7790.076} C_VEL
LIN {X 0,Y 482.637,Z 607.17,A -85,B 0,C 180,E1 7793.083,E2 7793.083} C_VEL
LIN {X 0,Y 480.435,Z 646.55,A -85,B 0,C 180,E1 7794.21,E2 7794.21} C_VEL
LIN {X 0,Y 475.721,Z 663.069,A -85,B 0,C 180,E1 7794.652,E2 7794.652} C_VEL
LIN {X 0,Y 470.876,Z 679.152,A -85,B 0,C 180,E1 7795.243,E2 7795.243} C_VEL
LIN {X 0,Y 467.222,Z 715.396,A -85,B 0,C 180,E1 7797.623,E2 7797.623} C_VEL
LIN {X 0,Y 463.186,Z 748.981,A -85,B 0,C 180,E1 7800.639,E2 7800.639} C_VEL
LIN {X 0,Y 459.268,Z 779.96,A -85,B 0,C 180,E1 7804.362,E2 7804.362} C_VEL
LIN {X 0,Y 456.061,Z 806.259,A -85,B 0,C 180,E1 7808.582,E2 7808.582} C_VEL
LIN {X 0,Y 453.89,Z 826.201,A -85,B 0,C 180,E1 7813.03,E2 7813.03} C_VEL
LIN {X 0,Y 452.626,Z 841.957,A -85,B 0,C 180,E1 7817.933,E2 7817.933} C_VEL
LIN {X 0,Y 452.198,Z 851.177,A -85,B 0,C 180,E1 7822.304,E2 7822.304} C_VEL
LIN {X 0,Y 452.059,Z 855.896,A -85,B 0,C 180,E1 7826.16,E2 7826.16} C_VEL
LIN {X 0,Y 452.079,Z 857.5,A -85,B 0,C 180,E1 7830,E2 7830} C_VEL
LIN {X 0,Y 452.042,Z 855.899,A -85,B 0,C 180,E1 7833.841,E2 7833.841} C_VEL
LIN {X 0,Y 452.316,Z 849.917,A -85,B 0,C 180,E1 7838.47,E2 7838.47} C_VEL
LIN {X 0,Y 452.987,Z 837.896,A -85,B 0,C 180,E1 7843.531,E2 7843.531} C_VEL
LIN {X 0,Y 454.551,Z 819.786,A -85,B 0,C 180,E1 7848.55,E2 7848.55} C_VEL
LIN {X 0,Y 456.947,Z 799.103,A -85,B 0,C 180,E1 7852.704,E2 7852.704} C_VEL
LIN {X 0,Y 460.395,Z 770.578,A -85,B 0,C 180,E1 7856.884,E2 7856.884} C_VEL
LIN {X 0,Y 464.26,Z 739.97,A -85,B 0,C 180,E1 7860.266,E2 7860.266} C_VEL
LIN {X 0,Y 468.239,Z 705.491,A -85,B 0,C 180,E1 7863.112,E2 7863.112} C_VEL
LIN {X 0,Y 471.97,Z 667.382,A -85,B 0,C 180,E1 7865.365,E2 7865.365} C_VEL
LIN {X 0,Y 474.778,Z 628.735,A -85,B 0,C 180,E1 7866.879,E2 7866.879} C_VEL
LIN {X 0,Y 475.259,Z 608.48,A -85,B 0,C 180,E1 7867.451,E2 7867.451} C_VEL
LIN {X 0,Y 450.838,Z 557.03,A -85,B 0,C 180,E1 7870.693,E2 7870.693} C_VEL
LIN {X 0,Y 450.891,Z 557.03,A -85,B 0,C 180,E1 7877.625,E2 7877.625} C_VEL
LIN {X 0,Y 450.89,Z 557.03,A -85,B 0,C 180,E1 7883.698,E2 7883.698} C_VEL
LIN {X 0,Y 450.948,Z 557.03,A -85,B 0,C 180,E1 7889.762,E2 7889.762} C_VEL
LIN {X 0,Y 451.15,Z 557.03,A -85,B 0,C 180,E1 7896.253,E2 7896.253} C_VEL
LIN {X 0,Y 451.299,Z 557.03,A -85,B 0,C 180,E1 7902.427,E2 7902.427} C_VEL
LIN {X 0,Y 451.346,Z 557.03,A -85,B 0,C 180,E1 7908.389,E2 7908.389} C_VEL
LIN {X 0,Y 451.725,Z 557.03,A -85,B 0,C 180,E1 7914.229,E2 7914.229} C_VEL
LIN {X 0,Y 451.926,Z 557.03,A -85,B 0,C 180,E1 7920,E2 7920} C_VEL
LIN {X 0,Y 451.666,Z 557.03,A -85,B 0,C 180,E1 7925.771,E2 7925.771} C_VEL
LIN {X 0,Y 451.456,Z 557.03,A -85,B 0,C 180,E1 7931.607,E2 7931.607} C_VEL
LIN {X 0,Y 451.346,Z 557.03,A -85,B 0,C 180,E1 7937.571,E2 7937.571} C_VEL
LIN {X 0,Y 451.146,Z 557.03,A -85,B 0,C 180,E1 7943.746,E2 7943.746} C_VEL
LIN {X 0,Y 450.956,Z 557.03,A -85,B 0,C 180,E1 7950.237,E2 7950.237} C_VEL
LIN {X 0,Y 450.851,Z 557.03,A -85,B 0,C 180,E1 7957.188,E2 7957.188} C_VEL
LIN {X 0,Y 450.786,Z 557.03,A -85,B 0,C 180,E1 7962.361,E2 7962.361} C_VEL
LIN {X 0,Y 450.889,Z 557.03,A -85,B 0,C 180,E1 7967.81,E2 7967.81} C_VEL
LIN {X 0,Y 450.905,Z 557.03,A -85,B 0,C 180,E1 7973.842,E2 7973.842} C_VEL
LIN {X 0,Y 455.279,Z 566.787,A -85,B 0,C 180,E1 7974.462,E2 7974.462} C_VEL
LIN {X 0,Y 474.049,Z 604.412,A -85,B 0,C 180,E1 7977.013,E2 7977.013} C_VEL
LIN {X 0,Y 471.601,Z 640.382,A -85,B 0,C 180,E1 7978.295,E2 7978.295} C_VEL
LIN {X 0,Y 468.088,Z 675.146,A -85,B 0,C 180,E1 7980.311,E2 7980.311} C_VEL
LIN {X 0,Y 464.213,Z 705.445,A -85,B 0,C 180,E1 7982.831,E2 7982.831} C_VEL
LIN {X 0,Y 460.299,Z 733.027,A -85,B 0,C 180,E1 7985.98,E2 7985.98} C_VEL
LIN {X 0,Y 456.68,Z 758.235,A -85,B 0,C 180,E1 7989.881,E2 7989.881} C_VEL
LIN {X 0,Y 454.268,Z 777.919,A -85,B 0,C 180,E1 7994.04,E2 7994.04} C_VEL
LIN {X 0,Y 452.858,Z 792.695,A -85,B 0,C 180,E1 7998.428,E2 7998.428} C_VEL
LIN {X 0,Y 452.38,Z 801.499,A -85,B 0,C 180,E1 8002.306,E2 8002.306} C_VEL
LIN {X 0,Y 452.15,Z 806.604,A -85,B 0,C 180,E1 8006.16,E2 8006.16} C_VEL
LIN {X 0,Y 452.121,Z 808.324,A -85,B 0,C 180,E1 8010,E2 8010} C_VEL
LIN {X 0,Y 452.253,Z 805.558,A -85,B 0,C 180,E1 8014.801,E2 8014.801} C_VEL
LIN {X 0,Y 452.607,Z 797.342,A -85,B 0,C 180,E1 8019.628,E2 8019.628} C_VEL
LIN {X 0,Y 453.731,Z 783.372,A -85,B 0,C 180,E1 8024.43,E2 8024.43} C_VEL
LIN {X 0,Y 455.926,Z 763.758,A -85,B 0,C 180,E1 8028.984,E2 8028.984} C_VEL
LIN {X 0,Y 459.262,Z 739.713,A -85,B 0,C 180,E1 8033.014,E2 8033.014} C_VEL
LIN {X 0,Y 463.501,Z 710.831,A -85,B 0,C 180,E1 8036.544,E2 8036.544} C_VEL
LIN {X 0,Y 467.643,Z 679.006,A -85,B 0,C 180,E1 8039.32,E2 8039.32} C_VEL
LIN {X 0,Y 471.152,Z 645.882,A -85,B 0,C 180,E1 8041.338,E2 8041.338} C_VEL
LIN {X 0,Y 473.686,Z 610.282,A -85,B 0,C 180,E1 8042.736,E2 8042.736} C_VEL
LIN {X 0,Y 473.21,Z 601.696,A -85,B 0,C 180,E1 8043.045,E2 8043.045} C_VEL
LIN {X 0,Y 451.017,Z 558.359,A -85,B 0,C 180,E1 8046.024,E2 8046.024} C_VEL
LIN {X 0,Y 450.875,Z 557.03,A -85,B 0,C 180,E1 8046.239,E2 8046.239} C_VEL
LIN {X 0,Y 450.833,Z 557.03,A -85,B 0,C 180,E1 8052.373,E2 8052.373} C_VEL
LIN {X 0,Y 450.891,Z 557.03,A -85,B 0,C 180,E1 8057.815,E2 8057.815} C_VEL
LIN {X 0,Y 450.868,Z 557.03,A -85,B 0,C 180,E1 8063.7,E2 8063.7} C_VEL
LIN {X 0,Y 450.94,Z 557.03,A -85,B 0,C 180,E1 8069.762,E2 8069.762} C_VEL
LIN {X 0,Y 451.162,Z 557.03,A -85,B 0,C 180,E1 8076.255,E2 8076.255} C_VEL
LIN {X 0,Y 451.415,Z 557.03,A -85,B 0,C 180,E1 8082.432,E2 8082.432} C_VEL
LIN {X 0,Y 451.513,Z 557.03,A -85,B 0,C 180,E1 8088.394,E2 8088.394} C_VEL
LIN {X 0,Y 451.665,Z 557.03,A -85,B 0,C 180,E1 8094.229,E2 8094.229} C_VEL
LIN {X 0,Y 451.939,Z 557.03,A -85,B 0,C 180,E1 8100,E2 8100} C_VEL
LIN {X 0,Y 451.724,Z 557.03,A -85,B 0,C 180,E1 8105.771,E2 8105.771} C_VEL
LIN {X 0,Y 451.444,Z 557.03,A -85,B 0,C 180,E1 8111.608,E2 8111.608} C_VEL
LIN {X 0,Y 451.277,Z 557.03,A -85,B 0,C 180,E1 8117.574,E2 8117.574} C_VEL
LIN {X 0,Y 451.152,Z 557.03,A -85,B 0,C 180,E1 8123.747,E2 8123.747} C_VEL
LIN {X 0,Y 450.945,Z 557.03,A -85,B 0,C 180,E1 8130.238,E2 8130.238} C_VEL
LIN {X 0,Y 450.896,Z 557.03,A -85,B 0,C 180,E1 8137.184,E2 8137.184} C_VEL
LIN {X 0,Y 450.892,Z 557.03,A -85,B 0,C 180,E1 8142.376,E2 8142.376} C_VEL
LIN {X 0,Y 450.891,Z 557.03,A -85,B 0,C 180,E1 8149.317,E2 8149.317} C_VEL
LIN {X 0,Y 457.15,Z 570.674,A -85,B 0,C 180,E1 8150.21,E2 8150.21} C_VEL
LIN {X 0,Y 475.845,Z 610.528,A -85,B 0,C 180,E1 8152.649,E2 8152.649} C_VEL
LIN {X 0,Y 473.287,Z 650.944,A -85,B 0,C 180,E1 8153.901,E2 8153.901} C_VEL
LIN {X 0,Y 470.876,Z 679.152,A -85,B 0,C 180,E1 8155.243,E2 8155.243} C_VEL
LIN {X 0,Y 465.815,Z 694.988,A -85,B 0,C 180,E1 8155.942,E2 8155.942} C_VEL
LIN {X 0,Y 460.936,Z 708.388,A -85,B 0,C 180,E1 8156.647,E2 8156.647} C_VEL
LIN {X 0,Y 460.656,Z 710.25,A -85,B 0,C 180,E1 8156.786,E2 8156.786} C_VEL
LIN {X 0,Y 456.219,Z 745.76,A -85,B 0,C 180,E1 8159.905,E2 8159.905} C_VEL
LIN {X 0,Y 452.291,Z 775.426,A -85,B 0,C 180,E1 8163.402,E2 8163.402} C_VEL
LIN {X 0,Y 448.874,Z 802.034,A -85,B 0,C 180,E1 8167.548,E2 8167.548} C_VEL
LIN {X 0,Y 446.652,Z 822.445,A -85,B 0,C 180,E1 8171.767,E2 8171.767} C_VEL
LIN {X 0,Y 444.974,Z 839.281,A -85,B 0,C 180,E1 8176.723,E2 8176.723} C_VEL
LIN {X 0,Y 444.449,Z 849.294,A -85,B 0,C 180,E1 8181.057,E2 8181.057} C_VEL
LIN {X 0,Y 444.152,Z 855.896,A -85,B 0,C 180,E1 8186.091,E2 8186.091} C_VEL
LIN {X 0,Y 444.179,Z 857.5,A -85,B 0,C 180,E1 8190,E2 8190} C_VEL
LIN {X 0,Y 444.138,Z 855.898,A -85,B 0,C 180,E1 8193.91,E2 8193.91} C_VEL
LIN {X 0,Y 444.464,Z 849.272,A -85,B 0,C 180,E1 8198.955,E2 8198.955} C_VEL
LIN {X 0,Y 445.166,Z 837.896,A -85,B 0,C 180,E1 8203.773,E2 8203.773} C_VEL
LIN {X 0,Y 446.731,Z 821.137,A -85,B 0,C 180,E1 8208.557,E2 8208.557} C_VEL
LIN {X 0,Y 449.335,Z 798.615,A -85,B 0,C 180,E1 8213.061,E2 8213.061} C_VEL
LIN {X 0,Y 452.92,Z 770.654,A -85,B 0,C 180,E1 8217.23,E2 8217.23} C_VEL
LIN {X 0,Y 457.01,Z 739.599,A -85,B 0,C 180,E1 8220.708,E2 8220.708} C_VEL
LIN {X 0,Y 461.323,Z 704.456,A -85,B 0,C 180,E1 8223.629,E2 8223.629} C_VEL
LIN {X 0,Y 465.146,Z 666.98,A -85,B 0,C 180,E1 8225.867,E2 8225.867} C_VEL
LIN {X 0,Y 468.155,Z 627.471,A -85,B 0,C 180,E1 8227.427,E2 8227.427} C_VEL
LIN {X 0,Y 468.514,Z 611.107,A -85,B 0,C 180,E1 8227.91,E2 8227.91} C_VEL
LIN {X 0,Y 444.885,Z 562.219,A -85,B 0,C 180,E1 8231.178,E2 8231.178} C_VEL
LIN {X 0,Y 442.903,Z 557.03,A -85,B 0,C 180,E1 8231.528,E2 8231.528} C_VEL
LIN {X 0,Y 442.891,Z 557.03,A -85,B 0,C 180,E1 8236.869,E2 8236.869} C_VEL
LIN {X 0,Y 442.926,Z 557.03,A -85,B 0,C 180,E1 8242.03,E2 8242.03} C_VEL
LIN {X 0,Y 442.954,Z 557.03,A -85,B 0,C 180,E1 8248.707,E2 8248.707} C_VEL
LIN {X 0,Y 443.145,Z 557.03,A -85,B 0,C 180,E1 8253.632,E2 8253.632} C_VEL
LIN {X 0,Y 443.368,Z 557.03,A -85,B 0,C 180,E1 8260.033,E2 8260.033} C_VEL
LIN {X 0,Y 443.333,Z 557.03,A -85,B 0,C 180,E1 8266.17,E2 8266.17} C_VEL
LIN {X 0,Y 443.697,Z 557.03,A -85,B 0,C 180,E1 8272.155,E2 8272.155} C_VEL
LIN {X 0,Y 444.049,Z 557.03,A -85,B 0,C 180,E1 8278.046,E2 8278.046} C_VEL
LIN {X 0,Y 443.964,Z 557.03,A -85,B 0,C 180,E1 8283.91,E2 8283.91} C_VEL
LIN {X 0,Y 443.658,Z 557.03,A -85,B 0,C 180,E1 8289.824,E2 8289.824} C_VEL
LIN {X 0,Y 443.441,Z 557.03,A -85,B 0,C 180,E1 8295.85,E2 8295.85} C_VEL
LIN {X 0,Y 443.264,Z 557.03,A -85,B 0,C 180,E1 8302.067,E2 8302.067} C_VEL
LIN {X 0,Y 443.046,Z 557.03,A -85,B 0,C 180,E1 8308.58,E2 8308.58} C_VEL
LIN {X 0,Y 442.92,Z 557.03,A -85,B 0,C 180,E1 8315.526,E2 8315.526} C_VEL
LIN {X 0,Y 442.804,Z 557.03,A -85,B 0,C 180,E1 8321.215,E2 8321.215} C_VEL
LIN {X 0,Y 442.886,Z 557.03,A -85,B 0,C 180,E1 8326.864,E2 8326.864} C_VEL
LIN {X 0,Y 443.024,Z 557.813,A -85,B 0,C 180,E1 8333.042,E2 8333.042} C_VEL
LIN {X 0,Y 467.348,Z 605.952,A -85,B 0,C 180,E1 8336.46,E2 8336.46} C_VEL
LIN {X 0,Y 464.824,Z 643.535,A -85,B 0,C 180,E1 8337.89,E2 8337.89} C_VEL
LIN {X 0,Y 461.317,Z 676.119,A -85,B 0,C 180,E1 8339.83,E2 8339.83} C_VEL
LIN {X 0,Y 457.058,Z 707.467,A -85,B 0,C 180,E1 8342.493,E2 8342.493} C_VEL
LIN {X 0,Y 452.815,Z 735.801,A -85,B 0,C 180,E1 8345.82,E2 8345.82} C_VEL
LIN {X 0,Y 449.035,Z 760.422,A -85,B 0,C 180,E1 8349.781,E2 8349.781} C_VEL
LIN {X 0,Y 446.393,Z 780.439,A -85,B 0,C 180,E1 8354.256,E2 8354.256} C_VEL
LIN {X 0,Y 444.962,Z 794.524,A -85,B 0,C 180,E1 8358.717,E2 8358.717} C_VEL
LIN {X 0,Y 444.461,Z 803.562,A -85,B 0,C 180,E1 8363.152,E2 8363.152} C_VEL
LIN {X 0,Y 444.231,Z 808.323,A -85,B 0,C 180,E1 8368.046,E2 8368.046} C_VEL
LIN {X 0,Y 444.26,Z 808.277,A -85,B 0,C 180,E1 8371.953,E2 8371.953} C_VEL
LIN {X 0,Y 444.464,Z 803.429,A -85,B 0,C 180,E1 8376.847,E2 8376.847} C_VEL
LIN {X 0,Y 445.143,Z 793.014,A -85,B 0,C 180,E1 8381.775,E2 8381.775} C_VEL
LIN {X 0,Y 446.911,Z 776.201,A -85,B 0,C 180,E1 8386.736,E2 8386.736} C_VEL
LIN {X 0,Y 449.761,Z 755.824,A -85,B 0,C 180,E1 8390.957,E2 8390.957} C_VEL
LIN {X 0,Y 453.475,Z 731.489,A -85,B 0,C 180,E1 8394.667,E2 8394.667} C_VEL
LIN {X 0,Y 457.889,Z 701.712,A -85,B 0,C 180,E1 8397.983,E2 8397.983} C_VEL
LIN {X 0,Y 462.034,Z 669.716,A -85,B 0,C 180,E1 8400.525,E2 8400.525} C_VEL
LIN {X 0,Y 465.623,Z 635.513,A -85,B 0,C 180,E1 8402.378,E2 8402.378} C_VEL
LIN {X 0,Y 466.869,Z 604.857,A -85,B 0,C 180,E1 8403.522,E2 8403.522} C_VEL
LIN {X 0,Y 444.405,Z 561.578,A -85,B 0,C 180,E1 8406.645,E2 8406.645} C_VEL
LIN {X 0,Y 442.979,Z 557.03,A -85,B 0,C 180,E1 8406.959,E2 8406.959} C_VEL
LIN {X 0,Y 442.892,Z 557.03,A -85,B 0,C 180,E1 8414.124,E2 8414.124} C_VEL
LIN {X 0,Y 442.901,Z 557.03,A -85,B 0,C 180,E1 8419.499,E2 8419.499} C_VEL
LIN {X 0,Y 442.944,Z 557.03,A -85,B 0,C 180,E1 8425.12,E2 8425.12} C_VEL
LIN {X 0,Y 443.049,Z 557.03,A -85,B 0,C 180,E1 8431.42,E2 8431.42} C_VEL
LIN {X 0,Y 443.292,Z 557.03,A -85,B 0,C 180,E1 8437.934,E2 8437.934} C_VEL
LIN {X 0,Y 443.52,Z 557.03,A -85,B 0,C 180,E1 8444.153,E2 8444.153} C_VEL
LIN {X 0,Y 443.69,Z 557.03,A -85,B 0,C 180,E1 8450.177,E2 8450.177} C_VEL
LIN {X 0,Y 443.961,Z 557.03,A -85,B 0,C 180,E1 8456.09,E2 8456.09} C_VEL
LIN {X 0,Y 444.043,Z 557.03,A -85,B 0,C 180,E1 8461.954,E2 8461.954} C_VEL
LIN {X 0,Y 443.649,Z 557.03,A -85,B 0,C 180,E1 8468.237,E2 8468.237} C_VEL
LIN {X 0,Y 443.463,Z 557.03,A -85,B 0,C 180,E1 8473.826,E2 8473.826} C_VEL
LIN {X 0,Y 443.319,Z 557.03,A -85,B 0,C 180,E1 8479.969,E2 8479.969} C_VEL
LIN {X 0,Y 443.145,Z 557.03,A -85,B 0,C 180,E1 8486.368,E2 8486.368} C_VEL
LIN {X 0,Y 442.959,Z 557.03,A -85,B 0,C 180,E1 8493.151,E2 8493.151} C_VEL
LIN {X 0,Y 442.918,Z 557.03,A -85,B 0,C 180,E1 8498.167,E2 8498.167} C_VEL
LIN {X 0,Y 442.915,Z 557.03,A -85,B 0,C 180,E1 8504.123,E2 8504.123} C_VEL
LIN {X 0,Y 442.993,Z 557.03,A -85,B 0,C 180,E1 8508.501,E2 8508.501} C_VEL
LIN {X 0,Y 452.022,Z 575.876,A -85,B 0,C 180,E1 8509.826,E2 8509.826} C_VEL
LIN {X 0,Y 469.097,Z 612.472,A -85,B 0,C 180,E1 8512.176,E2 8512.176} C_VEL
LIN {X 0,Y 466.362,Z 652.516,A -85,B 0,C 180,E1 8513.471,E2 8513.471} C_VEL
LIN {X 0,Y 462.721,Z 690.837,A -85,B 0,C 180,E1 8515.457,E2 8515.457} C_VEL
LIN {X 0,Y 460.656,Z 710.25,A -85,B 0,C 180,E1 8516.786,E2 8516.786} C_VEL
LIN {X 0,Y 455.344,Z 725.148,A -85,B 0,C 180,E1 8517.771,E2 8517.771} C_VEL
LIN {X 0,Y 449.771,Z 739.28,A -85,B 0,C 180,E1 8518.847,E2 8518.847} C_VEL
LIN {X 0,Y 445.202,Z 772.282,A -85,B 0,C 180,E1 8522.615,E2 8522.615} C_VEL
LIN {X 0,Y 441.361,Z 800.709,A -85,B 0,C 180,E1 8527.033,E2 8527.033} C_VEL
LIN {X 0,Y 438.851,Z 822.435,A -85,B 0,C 180,E1 8531.581,E2 8531.581} C_VEL
LIN {X 0,Y 437.166,Z 839.281,A -85,B 0,C 180,E1 8536.481,E2 8536.481} C_VEL
LIN {X 0,Y 436.566,Z 849.294,A -85,B 0,C 180,E1 8540.894,E2 8540.894} C_VEL
LIN {X 0,Y 436.245,Z 855.895,A -85,B 0,C 180,E1 8546.02,E2 8546.02} C_VEL
LIN {X 0,Y 436.278,Z 857.5,A -85,B 0,C 180,E1 8550,E2 8550} C_VEL
LIN {X 0,Y 436.234,Z 855.898,A -85,B 0,C 180,E1 8553.981,E2 8553.981} C_VEL
LIN {X 0,Y 436.576,Z 849.272,A -85,B 0,C 180,E1 8559.118,E2 8559.118} C_VEL
LIN {X 0,Y 437.463,Z 837.034,A -85,B 0,C 180,E1 8564.301,E2 8564.301} C_VEL
LIN {X 0,Y 439.045,Z 819.765,A -85,B 0,C 180,E1 8569.06,E2 8569.06} C_VEL
LIN {X 0,Y 441.956,Z 796.315,A -85,B 0,C 180,E1 8573.737,E2 8573.737} C_VEL
LIN {X 0,Y 445.606,Z 769.515,A -85,B 0,C 180,E1 8577.736,E2 8577.736} C_VEL
LIN {X 0,Y 449.819,Z 738.91,A -85,B 0,C 180,E1 8581.188,E2 8581.188} C_VEL
LIN {X 0,Y 454.344,Z 703.874,A -85,B 0,C 180,E1 8584.132,E2 8584.132} C_VEL
LIN {X 0,Y 458.412,Z 666.275,A -85,B 0,C 180,E1 8586.402,E2 8586.402} C_VEL
LIN {X 0,Y 461.625,Z 627.053,A -85,B 0,C 180,E1 8587.978,E2 8587.978} C_VEL
LIN {X 0,Y 461.823,Z 613.756,A -85,B 0,C 180,E1 8588.4,E2 8588.4} C_VEL
LIN {X 0,Y 439.624,Z 567.185,A -85,B 0,C 180,E1 8591.619,E2 8591.619} C_VEL
LIN {X 0,Y 435.011,Z 557.03,A -85,B 0,C 180,E1 8592.414,E2 8592.414} C_VEL
LIN {X 0,Y 434.993,Z 557.03,A -85,B 0,C 180,E1 8598.602,E2 8598.602} C_VEL
LIN {X 0,Y 434.952,Z 557.03,A -85,B 0,C 180,E1 8603.72,E2 8603.72} C_VEL
LIN {X 0,Y 435.051,Z 557.03,A -85,B 0,C 180,E1 8608.534,E2 8608.534} C_VEL
LIN {X 0,Y 435.25,Z 557.03,A -85,B 0,C 180,E1 8615.329,E2 8615.329} C_VEL
LIN {X 0,Y 435.44,Z 557.03,A -85,B 0,C 180,E1 8621.765,E2 8621.765} C_VEL
LIN {X 0,Y 435.489,Z 557.03,A -85,B 0,C 180,E1 8627.96,E2 8627.96} C_VEL
LIN {X 0,Y 435.886,Z 557.03,A -85,B 0,C 180,E1 8634.019,E2 8634.019} C_VEL
LIN {X 0,Y 436.133,Z 557.03,A -85,B 0,C 180,E1 8640,E2 8640} C_VEL
LIN {X 0,Y 435.833,Z 557.03,A -85,B 0,C 180,E1 8645.981,E2 8645.981} C_VEL
LIN {X 0,Y 435.601,Z 557.03,A -85,B 0,C 180,E1 8652.036,E2 8652.036} C_VEL
LIN {X 0,Y 435.465,Z 557.03,A -85,B 0,C 180,E1 8658.233,E2 8658.233} C_VEL
LIN {X 0,Y 435.203,Z 557.03,A -85,B 0,C 180,E1 8665.239,E2 8665.239} C_VEL
LIN {X 0,Y 435.059,Z 557.03,A -85,B 0,C 180,E1 8671.465,E2 8671.465} C_VEL
LIN {X 0,Y 434.895,Z 557.03,A -85,B 0,C 180,E1 8676.8,E2 8676.8} C_VEL
LIN {X 0,Y 434.903,Z 557.03,A -85,B 0,C 180,E1 8683.022,E2 8683.022} C_VEL
LIN {X 0,Y 434.987,Z 557.03,A -85,B 0,C 180,E1 8688.598,E2 8688.598} C_VEL
LIN {X 0,Y 435.051,Z 557.03,A -85,B 0,C 180,E1 8692.127,E2 8692.127} C_VEL
LIN {X 0,Y 439.621,Z 566.999,A -85,B 0,C 180,E1 8692.854,E2 8692.854} C_VEL
LIN {X 0,Y 460.738,Z 608.519,A -85,B 0,C 180,E1 8695.942,E2 8695.942} C_VEL
LIN {X 0,Y 458.192,Z 645.012,A -85,B 0,C 180,E1 8697.388,E2 8697.388} C_VEL
LIN {X 0,Y 454.302,Z 678.693,A -85,B 0,C 180,E1 8699.453,E2 8699.453} C_VEL
LIN {X 0,Y 449.9,Z 709.582,A -85,B 0,C 180,E1 8702.164,E2 8702.164} C_VEL
LIN {X 0,Y 445.306,Z 738.375,A -85,B 0,C 180,E1 8705.653,E2 8705.653} C_VEL
LIN {X 0,Y 441.385,Z 762.451,A -85,B 0,C 180,E1 8709.677,E2 8709.677} C_VEL
LIN {X 0,Y 438.735,Z 781.114,A -85,B 0,C 180,E1 8713.973,E2 8713.973} C_VEL
LIN {X 0,Y 437.065,Z 796.356,A -85,B 0,C 180,E1 8719.016,E2 8719.016} C_VEL
LIN {X 0,Y 436.491,Z 805.449,A -85,B 0,C 180,E1 8724.027,E2 8724.027} C_VEL
LIN {X 0,Y 436.342,Z 808.77,A -85,B 0,C 180,E1 8728.011,E2 8728.011} C_VEL
LIN {X 0,Y 436.371,Z 808.723,A -85,B 0,C 180,E1 8731.988,E2 8731.988} C_VEL
LIN {X 0,Y 436.606,Z 803.912,A -85,B 0,C 180,E1 8736.971,E2 8736.971} C_VEL
LIN {X 0,Y 437.356,Z 793.586,A -85,B 0,C 180,E1 8741.988,E2 8741.988} C_VEL
LIN {X 0,Y 439.275,Z 776.911,A -85,B 0,C 180,E1 8747.035,E2 8747.035} C_VEL
LIN {X 0,Y 442.361,Z 756.603,A -85,B 0,C 180,E1 8751.325,E2 8751.325} C_VEL
LIN {X 0,Y 446.294,Z 732.241,A -85,B 0,C 180,E1 8755.091,E2 8755.091} C_VEL
LIN {X 0,Y 450.983,Z 702.371,A -85,B 0,C 180,E1 8758.469,E2 8758.469} C_VEL
LIN {X 0,Y 455.526,Z 668.83,A -85,B 0,C 180,E1 8761.148,E2 8761.148} C_VEL
LIN {X 0,Y 459.281,Z 633.908,A -85,B 0,C 180,E1 8763.027,E2 8763.027} C_VEL
LIN {X 0,Y 460.573,Z 608.008,A -85,B 0,C 180,E1 8763.999,E2 8763.999} C_VEL
LIN {X 0,Y 439.493,Z 566.815,A -85,B 0,C 180,E1 8767.067,E2 8767.067} C_VEL
LIN {X 0,Y 435.012,Z 557.03,A -85,B 0,C 180,E1 8767.872,E2 8767.872} C_VEL
LIN {X 0,Y 434.992,Z 557.03,A -85,B 0,C 180,E1 8774.117,E2 8774.117} C_VEL
LIN {X 0,Y 434.955,Z 557.03,A -85,B 0,C 180,E1 8779.978,E2 8779.978} C_VEL
LIN {X 0,Y 435.042,Z 557.03,A -85,B 0,C 180,E1 8786.642,E2 8786.642} C_VEL
LIN {X 0,Y 435.199,Z 557.03,A -85,B 0,C 180,E1 8793.113,E2 8793.113} C_VEL
LIN {X 0,Y 435.479,Z 557.03,A -85,B 0,C 180,E1 8799.837,E2 8799.837} C_VEL
LIN {X 0,Y 435.654,Z 557.03,A -85,B 0,C 180,E1 8805.921,E2 8805.921} C_VEL
LIN {X 0,Y 435.807,Z 557.03,A -85,B 0,C 180,E1 8812.013,E2 8812.013} C_VEL
LIN {X 0,Y 436.047,Z 557.03,A -85,B 0,C 180,E1 8818.011,E2 8818.011} C_VEL
LIN {X 0,Y 435.868,Z 557.03,A -85,B 0,C 180,E1 8823.984,E2 8823.984} C_VEL
LIN {X 0,Y 435.666,Z 557.03,A -85,B 0,C 180,E1 8830.006,E2 8830.006} C_VEL
LIN {X 0,Y 435.465,Z 557.03,A -85,B 0,C 180,E1 8836.149,E2 8836.149} C_VEL
LIN {X 0,Y 435.321,Z 557.03,A -85,B 0,C 180,E1 8842.492,E2 8842.492} C_VEL
LIN {X 0,Y 435.062,Z 557.03,A -85,B 0,C 180,E1 8849.156,E2 8849.156} C_VEL
LIN {X 0,Y 435.029,Z 557.03,A -85,B 0,C 180,E1 8853.836,E2 8853.836} C_VEL
LIN {X 0,Y 434.962,Z 557.03,A -85,B 0,C 180,E1 8860.023,E2 8860.023} C_VEL
LIN {X 0,Y 434.996,Z 557.03,A -85,B 0,C 180,E1 8865.884,E2 8865.884} C_VEL
LIN {X 0,Y 435.065,Z 557.03,A -85,B 0,C 180,E1 8867.649,E2 8867.649} C_VEL
LIN {X 0,Y 439.673,Z 567.138,A -85,B 0,C 180,E1 8868.389,E2 8868.389} C_VEL
LIN {X 0,Y 462.129,Z 614.424,A -85,B 0,C 180,E1 8871.647,E2 8871.647} C_VEL
LIN {X 0,Y 459.406,Z 654.978,A -85,B 0,C 180,E1 8873.06,E2 8873.06} C_VEL
LIN {X 0,Y 455.4,Z 694.323,A -85,B 0,C 180,E1 8875.204,E2 8875.204} C_VEL
LIN {X 0,Y 450.837,Z 731.437,A -85,B 0,C 180,E1 8878.096,E2 8878.096} C_VEL
LIN {X 0,Y 449.771,Z 739.28,A -85,B 0,C 180,E1 8878.847,E2 8878.847} C_VEL
LIN {X 0,Y 444.26,Z 752.951,A -85,B 0,C 180,E1 8880.069,E2 8880.069} C_VEL
LIN {X 0,Y 438.692,Z 765.881,A -85,B 0,C 180,E1 8881.429,E2 8881.429} C_VEL
LIN {X 0,Y 434.608,Z 793.994,A -85,B 0,C 180,E1 8885.563,E2 8885.563} C_VEL
LIN {X 0,Y 431.654,Z 816.582,A -85,B 0,C 180,E1 8890.003,E2 8890.003} C_VEL
LIN {X 0,Y 429.792,Z 834.164,A -85,B 0,C 180,E1 8894.681,E2 8894.681} C_VEL
LIN {X 0,Y 428.794,Z 847.489,A -85,B 0,C 180,E1 8899.832,E2 8899.832} C_VEL
LIN {X 0,Y 428.414,Z 853.929,A -85,B 0,C 180,E1 8903.914,E2 8903.914} C_VEL
LIN {X 0,Y 428.364,Z 857.086,A -85,B 0,C 180,E1 8907.975,E2 8907.975} C_VEL
LIN {X 0,Y 428.394,Z 857.086,A -85,B 0,C 180,E1 8912.026,E2 8912.026} C_VEL
LIN {X 0,Y 428.508,Z 852.723,A -85,B 0,C 180,E1 8917.104,E2 8917.104} C_VEL
LIN {X 0,Y 429.047,Z 842.905,A -85,B 0,C 180,E1 8922.224,E2 8922.224} C_VEL
LIN {X 0,Y 430.49,Z 827.116,A -85,B 0,C 180,E1 8927.395,E2 8927.395} C_VEL
LIN {X 0,Y 433.037,Z 805.59,A -85,B 0,C 180,E1 8932.33,E2 8932.33} C_VEL
LIN {X 0,Y 436.754,Z 779.027,A -85,B 0,C 180,E1 8936.786,E2 8936.786} C_VEL
LIN {X 0,Y 441.081,Z 749.038,A -85,B 0,C 180,E1 8940.561,E2 8940.561} C_VEL
LIN {X 0,Y 445.77,Z 715.325,A -85,B 0,C 180,E1 8943.736,E2 8943.736} C_VEL
LIN {X 0,Y 450.333,Z 678.057,A -85,B 0,C 180,E1 8946.311,E2 8946.311} C_VEL
LIN {X 0,Y 454.283,Z 638.398,A -85,B 0,C 180,E1 8948.16,E2 8948.16} C_VEL
LIN {X 0,Y 455.277,Z 616.485,A -85,B 0,C 180,E1 8948.9,E2 8948.9} C_VEL
LIN {X 0,Y 434.756,Z 572.593,A -85,B 0,C 180,E1 8952.022,E2 8952.022} C_VEL
LIN {X 0,Y 427.14,Z 558.195,A -85,B 0,C 180,E1 8953.201,E2 8953.201} C_VEL
LIN {X 0,Y 427.045,Z 557.03,A -85,B 0,C 180,E1 8953.246,E2 8953.246} C_VEL
LIN {X 0,Y 427.056,Z 557.03,A -85,B 0,C 180,E1 8960.348,E2 8960.348} C_VEL
LIN {X 0,Y 427.026,Z 557.03,A -85,B 0,C 180,E1 8965.441,E2 8965.441} C_VEL
LIN {X 0,Y 427.208,Z 557.03,A -85,B 0,C 180,E1 8972.377,E2 8972.377} C_VEL
LIN {X 0,Y 427.46,Z 557.03,A -85,B 0,C 180,E1 8979.257,E2 8979.257} C_VEL
LIN {X 0,Y 427.498,Z 557.03,A -85,B 0,C 180,E1 8985.646,E2 8985.646} C_VEL
LIN {X 0,Y 427.879,Z 557.03,A -85,B 0,C 180,E1 8992.217,E2 8992.217} C_VEL
LIN {X 0,Y 428.251,Z 557.03,A -85,B 0,C 180,E1 8997.974,E2 8997.974} C_VEL
LIN {X 0,Y 428.125,Z 557.03,A -85,B 0,C 180,E1 9004.055,E2 9004.055} C_VEL
LIN {X 0,Y 427.789,Z 557.03,A -85,B 0,C 180,E1 9010.192,E2 9010.192} C_VEL
LIN {X 0,Y 427.55,Z 557.03,A -85,B 0,C 180,E1 9017.033,E2 9017.033} C_VEL
LIN {X 0,Y 427.391,Z 557.03,A -85,B 0,C 180,E1 9022.932,E2 9022.932} C_VEL
LIN {X 0,Y 427.155,Z 557.03,A -85,B 0,C 180,E1 9029.748,E2 9029.748} C_VEL
LIN {X 0,Y 426.964,Z 557.03,A -85,B 0,C 180,E1 9037.07,E2 9037.07} C_VEL
LIN {X 0,Y 426.966,Z 557.03,A -85,B 0,C 180,E1 9042.353,E2 9042.353} C_VEL
LIN {X 0,Y 427.067,Z 557.03,A -85,B 0,C 180,E1 9048.111,E2 9048.111} C_VEL
LIN {X 0,Y 427.062,Z 557.237,A -85,B 0,C 180,E1 9051.251,E2 9051.251} C_VEL
LIN {X 0,Y 431.525,Z 566.661,A -85,B 0,C 180,E1 9051.954,E2 9051.954} C_VEL
LIN {X 0,Y 452.676,Z 607.55,A -85,B 0,C 180,E1 9055.139,E2 9055.139} C_VEL
LIN {X 0,Y 454.384,Z 613.927,A -85,B 0,C 180,E1 9055.541,E2 9055.541} C_VEL
LIN {X 0,Y 451.393,Z 648.528,A -85,B 0,C 180,E1 9056.98,E2 9056.98} C_VEL
LIN {X 0,Y 447.096,Z 682.887,A -85,B 0,C 180,E1 9059.189,E2 9059.189} C_VEL
LIN {X 0,Y 442.281,Z 714.432,A -85,B 0,C 180,E1 9062.128,E2 9062.128} C_VEL
LIN {X 0,Y 437.575,Z 741.76,A -85,B 0,C 180,E1 9065.634,E2 9065.634} C_VEL
LIN {X 0,Y 433.542,Z 765.388,A -85,B 0,C 180,E1 9069.776,E2 9069.776} C_VEL
LIN {X 0,Y 430.752,Z 784.25,A -85,B 0,C 180,E1 9074.372,E2 9074.372} C_VEL
LIN {X 0,Y 429.175,Z 798.043,A -85,B 0,C 180,E1 9079.326,E2 9079.326} C_VEL
LIN {X 0,Y 428.62,Z 805.922,A -85,B 0,C 180,E1 9083.916,E2 9083.916} C_VEL
LIN {X 0,Y 428.453,Z 809.216,A -85,B 0,C 180,E1 9087.975,E2 9087.975} C_VEL
LIN {X 0,Y 428.481,Z 809.172,A -85,B 0,C 180,E1 9092.025,E2 9092.025} C_VEL
LIN {X 0,Y 428.743,Z 804.407,A -85,B 0,C 180,E1 9097.099,E2 9097.099} C_VEL
LIN {X 0,Y 429.598,Z 794.159,A -85,B 0,C 180,E1 9102.208,E2 9102.208} C_VEL
LIN {X 0,Y 431.544,Z 778.603,A -85,B 0,C 180,E1 9107.087,E2 9107.087} C_VEL
LIN {X 0,Y 434.729,Z 758.655,A -85,B 0,C 180,E1 9111.45,E2 9111.45} C_VEL
LIN {X 0,Y 438.773,Z 734.779,A -85,B 0,C 180,E1 9115.278,E2 9115.278} C_VEL
LIN {X 0,Y 443.423,Z 707.065,A -85,B 0,C 180,E1 9118.556,E2 9118.556} C_VEL
LIN {X 0,Y 448.158,Z 675.132,A -85,B 0,C 180,E1 9121.293,E2 9121.293} C_VEL
LIN {X 0,Y 452.369,Z 639.614,A -85,B 0,C 180,E1 9123.366,E2 9123.366} C_VEL
LIN {X 0,Y 453.889,Z 610.353,A -85,B 0,C 180,E1 9124.546,E2 9124.546} C_VEL
LIN {X 0,Y 434.28,Z 571.591,A -85,B 0,C 180,E1 9127.543,E2 9127.543} C_VEL
LIN {X 0,Y 427.179,Z 558.496,A -85,B 0,C 180,E1 9128.611,E2 9128.611} C_VEL
LIN {X 0,Y 427.021,Z 557.03,A -85,B 0,C 180,E1 9128.742,E2 9128.742} C_VEL
LIN {X 0,Y 427.059,Z 557.03,A -85,B 0,C 180,E1 9135.158,E2 9135.158} C_VEL
LIN {X 0,Y 427.039,Z 557.03,A -85,B 0,C 180,E1 9141.26,E2 9141.26} C_VEL
LIN {X 0,Y 427.131,Z 557.03,A -85,B 0,C 180,E1 9148.29,E2 9148.29} C_VEL
LIN {X 0,Y 427.332,Z 557.03,A -85,B 0,C 180,E1 9154.841,E2 9154.841} C_VEL
LIN {X 0,Y 427.591,Z 557.03,A -85,B 0,C 180,E1 9161.419,E2 9161.419} C_VEL
LIN {X 0,Y 427.766,Z 557.03,A -85,B 0,C 180,E1 9167.74,E2 9167.74} C_VEL
LIN {X 0,Y 427.918,Z 557.03,A -85,B 0,C 180,E1 9173.908,E2 9173.908} C_VEL
LIN {X 0,Y 428.243,Z 557.03,A -85,B 0,C 180,E1 9180,E2 9180} C_VEL
LIN {X 0,Y 427.966,Z 557.03,A -85,B 0,C 180,E1 9186.092,E2 9186.092} C_VEL
LIN {X 0,Y 427.664,Z 557.03,A -85,B 0,C 180,E1 9192.264,E2 9192.264} C_VEL
LIN {X 0,Y 427.475,Z 557.03,A -85,B 0,C 180,E1 9198.587,E2 9198.587} C_VEL
LIN {X 0,Y 427.325,Z 557.03,A -85,B 0,C 180,E1 9205.16,E2 9205.16} C_VEL
LIN {X 0,Y 427.098,Z 557.03,A -85,B 0,C 180,E1 9212.121,E2 9212.121} C_VEL
LIN {X 0,Y 427.049,Z 557.03,A -85,B 0,C 180,E1 9218.742,E2 9218.742} C_VEL
LIN {X 0,Y 427.06,Z 557.03,A -85,B 0,C 180,E1 9225.155,E2 9225.155} C_VEL
LIN {X 0,Y 427.083,Z 557.03,A -85,B 0,C 180,E1 9226.757,E2 9226.757} C_VEL
LIN {X 0,Y 431.385,Z 566.549,A -85,B 0,C 180,E1 9227.476,E2 9227.476} C_VEL
LIN {X 0,Y 448.377,Z 600.719,A -85,B 0,C 180,E1 9230.01,E2 9230.01} C_VEL
LIN {X 0,Y 455.727,Z 619.159,A -85,B 0,C 180,E1 9231.224,E2 9231.224} C_VEL
LIN {X 0,Y 452.192,Z 660.832,A -85,B 0,C 180,E1 9232.776,E2 9232.776} C_VEL
LIN {X 0,Y 447.841,Z 699.738,A -85,B 0,C 180,E1 9235.083,E2 9235.083} C_VEL
LIN {X 0,Y 443.11,Z 735.185,A -85,B 0,C 180,E1 9238.022,E2 9238.022} C_VEL
LIN {X 0,Y 438.692,Z 765.881,A -85,B 0,C 180,E1 9241.429,E2 9241.429} C_VEL
LIN {X 0,Y 433.073,Z 778.181,A -85,B 0,C 180,E1 9242.914,E2 9242.914} C_VEL
LIN {X 0,Y 427.554,Z 789.667,A -85,B 0,C 180,E1 9244.511,E2 9244.511} C_VEL
LIN {X 0,Y 424.07,Z 814.766,A -85,B 0,C 180,E1 9249.356,E2 9249.356} C_VEL
LIN {X 0,Y 421.996,Z 833.592,A -85,B 0,C 180,E1 9254.39,E2 9254.39} C_VEL
LIN {X 0,Y 420.911,Z 846.991,A -85,B 0,C 180,E1 9259.639,E2 9259.639} C_VEL
LIN {X 0,Y 420.425,Z 854.722,A -85,B 0,C 180,E1 9264.835,E2 9264.835} C_VEL
LIN {X 0,Y 420.502,Z 857.295,A -85,B 0,C 180,E1 9270,E2 9270} C_VEL
LIN {X 0,Y 420.442,Z 854.725,A -85,B 0,C 180,E1 9275.166,E2 9275.166} C_VEL
LIN {X 0,Y 420.875,Z 846.983,A -85,B 0,C 180,E1 9280.363,E2 9280.363} C_VEL
LIN {X 0,Y 421.948,Z 833.582,A -85,B 0,C 180,E1 9285.612,E2 9285.612} C_VEL
LIN {X 0,Y 424.067,Z 814.759,A -85,B 0,C 180,E1 9290.645,E2 9290.645} C_VEL
LIN {X 0,Y 427.537,Z 789.901,A -85,B 0,C 180,E1 9295.45,E2 9295.45} C_VEL
LIN {X 0,Y 432.245,Z 759.313,A -85,B 0,C 180,E1 9299.787,E2 9299.787} C_VEL
LIN {X 0,Y 437.263,Z 725.609,A -85,B 0,C 180,E1 9303.346,E2 9303.346} C_VEL
LIN {X 0,Y 442.275,Z 689.927,A -85,B 0,C 180,E1 9306.118,E2 9306.118} C_VEL
LIN {X 0,Y 446.52,Z 653.114,A -85,B 0,C 180,E1 9308.134,E2 9308.134} C_VEL
LIN {X 0,Y 448.885,Z 619.606,A -85,B 0,C 180,E1 9309.395,E2 9309.395} C_VEL
LIN {X 0,Y 430.534,Z 579.457,A -85,B 0,C 180,E1 9312.331,E2 9312.331} C_VEL
LIN {X 0,Y 419.237,Z 558.141,A -85,B 0,C 180,E1 9314.141,E2 9314.141} C_VEL
LIN {X 0,Y 419.14,Z 557.03,A -85,B 0,C 180,E1 9314.283,E2 9314.283} C_VEL
LIN {X 0,Y 419.086,Z 557.03,A -85,B 0,C 180,E1 9319.439,E2 9319.439} C_VEL
LIN {X 0,Y 419.08,Z 557.03,A -85,B 0,C 180,E1 9326.196,E2 9326.196} C_VEL
LIN {X 0,Y 419.264,Z 557.03,A -85,B 0,C 180,E1 9332.003,E2 9332.003} C_VEL
LIN {X 0,Y 419.522,Z 557.03,A -85,B 0,C 180,E1 9338.846,E2 9338.846} C_VEL
LIN {X 0,Y 419.564,Z 557.03,A -85,B 0,C 180,E1 9345.369,E2 9345.369} C_VEL
LIN {X 0,Y 419.935,Z 557.03,A -85,B 0,C 180,E1 9351.708,E2 9351.708} C_VEL
LIN {X 0,Y 420.336,Z 557.03,A -85,B 0,C 180,E1 9357.936,E2 9357.936} C_VEL
LIN {X 0,Y 420.205,Z 557.03,A -85,B 0,C 180,E1 9364.132,E2 9364.132} C_VEL
LIN {X 0,Y 419.854,Z 557.03,A -85,B 0,C 180,E1 9370.387,E2 9370.387} C_VEL
LIN {X 0,Y 419.696,Z 557.03,A -85,B 0,C 180,E1 9376.773,E2 9376.773} C_VEL
LIN {X 0,Y 419.423,Z 557.03,A -85,B 0,C 180,E1 9383.394,E2 9383.394} C_VEL
LIN {X 0,Y 419.211,Z 557.03,A -85,B 0,C 180,E1 9390.371,E2 9390.371} C_VEL
LIN {X 0,Y 419.06,Z 557.03,A -85,B 0,C 180,E1 9397.358,E2 9397.358} C_VEL
LIN {X 0,Y 419.008,Z 557.03,A -85,B 0,C 180,E1 9403.723,E2 9403.723} C_VEL
LIN {X 0,Y 419.162,Z 557.03,A -85,B 0,C 180,E1 9410.278,E2 9410.278} C_VEL
LIN {X 0,Y 421.675,Z 562.822,A -85,B 0,C 180,E1 9410.725,E2 9410.725} C_VEL
LIN {X 0,Y 444.467,Z 606.336,A -85,B 0,C 180,E1 9414.282,E2 9414.282} C_VEL
LIN {X 0,Y 447.969,Z 615.484,A -85,B 0,C 180,E1 9414.976,E2 9414.976} C_VEL
LIN {X 0,Y 444.645,Z 651.551,A -85,B 0,C 180,E1 9416.533,E2 9416.533} C_VEL
LIN {X 0,Y 439.89,Z 686.722,A -85,B 0,C 180,E1 9418.916,E2 9418.916} C_VEL
LIN {X 0,Y 434.786,Z 717.906,A -85,B 0,C 180,E1 9421.958,E2 9421.958} C_VEL
LIN {X 0,Y 429.87,Z 744.758,A -85,B 0,C 180,E1 9425.558,E2 9425.558} C_VEL
LIN {X 0,Y 425.732,Z 768.105,A -85,B 0,C 180,E1 9429.851,E2 9429.851} C_VEL
LIN {X 0,Y 422.863,Z 786.24,A -85,B 0,C 180,E1 9434.529,E2 9434.529} C_VEL
LIN {X 0,Y 421.334,Z 799.652,A -85,B 0,C 180,E1 9439.649,E2 9439.649} C_VEL
LIN {X 0,Y 420.73,Z 807.534,A -85,B 0,C 180,E1 9444.838,E2 9444.838} C_VEL
LIN {X 0,Y 420.618,Z 810.092,A -85,B 0,C 180,E1 9450,E2 9450} C_VEL
LIN {X 0,Y 420.755,Z 807.43,A -85,B 0,C 180,E1 9455.161,E2 9455.161} C_VEL
LIN {X 0,Y 421.327,Z 799.468,A -85,B 0,C 180,E1 9460.351,E2 9460.351} C_VEL
LIN {X 0,Y 422.991,Z 785.629,A -85,B 0,C 180,E1 9465.571,E2 9465.571} C_VEL
LIN {X 0,Y 426.081,Z 766.059,A -85,B 0,C 180,E1 9470.485,E2 9470.485} C_VEL
LIN {X 0,Y 430.33,Z 742.316,A -85,B 0,C 180,E1 9474.723,E2 9474.723} C_VEL
LIN {X 0,Y 435.252,Z 714.949,A -85,B 0,C 180,E1 9478.291,E2 9478.291} C_VEL
LIN {X 0,Y 440.561,Z 682.641,A -85,B 0,C 180,E1 9481.318,E2 9481.318} C_VEL
LIN {X 0,Y 444.898,Z 649.162,A -85,B 0,C 180,E1 9483.497,E2 9483.497} C_VEL
LIN {X 0,Y 447.501,Z 613.154,A -85,B 0,C 180,E1 9485.065,E2 9485.065} C_VEL
LIN {X 0,Y 429.48,Z 576.926,A -85,B 0,C 180,E1 9487.975,E2 9487.975} C_VEL
LIN {X 0,Y 419.15,Z 557.735,A -85,B 0,C 180,E1 9489.589,E2 9489.589} C_VEL
LIN {X 0,Y 419.064,Z 557.03,A -85,B 0,C 180,E1 9496.654,E2 9496.654} C_VEL
LIN {X 0,Y 419.089,Z 557.03,A -85,B 0,C 180,E1 9502.636,E2 9502.636} C_VEL
LIN {X 0,Y 419.255,Z 557.03,A -85,B 0,C 180,E1 9510.078,E2 9510.078} C_VEL
LIN {X 0,Y 419.425,Z 557.03,A -85,B 0,C 180,E1 9516.606,E2 9516.606} C_VEL
LIN {X 0,Y 419.761,Z 557.03,A -85,B 0,C 180,E1 9523.23,E2 9523.23} C_VEL
LIN {X 0,Y 419.901,Z 557.03,A -85,B 0,C 180,E1 9529.615,E2 9529.615} C_VEL
LIN {X 0,Y 420.202,Z 557.03,A -85,B 0,C 180,E1 9535.868,E2 9535.868} C_VEL
LIN {X 0,Y 420.33,Z 557.03,A -85,B 0,C 180,E1 9542.064,E2 9542.064} C_VEL
LIN {X 0,Y 419.952,Z 557.03,A -85,B 0,C 180,E1 9548.291,E2 9548.291} C_VEL
LIN {X 0,Y 419.676,Z 557.03,A -85,B 0,C 180,E1 9554.627,E2 9554.627} C_VEL
LIN {X 0,Y 419.484,Z 557.03,A -85,B 0,C 180,E1 9561.156,E2 9561.156} C_VEL
LIN {X 0,Y 419.263,Z 557.03,A -85,B 0,C 180,E1 9567.997,E2 9567.997} C_VEL
LIN {X 0,Y 419.104,Z 557.03,A -85,B 0,C 180,E1 9575.309,E2 9575.309} C_VEL
LIN {X 0,Y 419.083,Z 557.03,A -85,B 0,C 180,E1 9580.653,E2 9580.653} C_VEL
LIN {X 0,Y 419.196,Z 557.03,A -85,B 0,C 180,E1 9585.817,E2 9585.817} C_VEL
LIN {X 0,Y 423.741,Z 567.019,A -85,B 0,C 180,E1 9586.614,E2 9586.614} C_VEL
LIN {X 0,Y 441.016,Z 601.012,A -85,B 0,C 180,E1 9589.286,E2 9589.286} C_VEL
LIN {X 0,Y 449.232,Z 620.348,A -85,B 0,C 180,E1 9590.662,E2 9590.662} C_VEL
LIN {X 0,Y 445.444,Z 662.215,A -85,B 0,C 180,E1 9592.28,E2 9592.28} C_VEL
LIN {X 0,Y 440.976,Z 699.719,A -85,B 0,C 180,E1 9594.553,E2 9594.553} C_VEL
LIN {X 0,Y 435.912,Z 735.262,A -85,B 0,C 180,E1 9597.576,E2 9597.576} C_VEL
LIN {X 0,Y 431.133,Z 766.715,A -85,B 0,C 180,E1 9601.152,E2 9601.152} C_VEL
LIN {X 0,Y 427.554,Z 789.667,A -85,B 0,C 180,E1 9604.511,E2 9604.511} C_VEL
LIN {X 0,Y 422.222,Z 800.35,A -85,B 0,C 180,E1 9606.243,E2 9606.243} C_VEL
LIN {X 0,Y 416.924,Z 810.161,A -85,B 0,C 180,E1 9608.101,E2 9608.101} C_VEL
LIN {X 0,Y 414.476,Z 829.537,A -85,B 0,C 180,E1 9613.009,E2 9613.009} C_VEL
LIN {X 0,Y 413.202,Z 843.062,A -85,B 0,C 180,E1 9617.838,E2 9617.838} C_VEL
LIN {X 0,Y 412.716,Z 852.124,A -85,B 0,C 180,E1 9622.855,E2 9622.855} C_VEL
LIN {X 0,Y 412.565,Z 856.415,A -85,B 0,C 180,E1 9627.897,E2 9627.897} C_VEL
LIN {X 0,Y 412.593,Z 856.417,A -85,B 0,C 180,E1 9632.103,E2 9632.103} C_VEL
LIN {X 0,Y 412.741,Z 852.123,A -85,B 0,C 180,E1 9637.15,E2 9637.15} C_VEL
LIN {X 0,Y 413.357,Z 841.86,A -85,B 0,C 180,E1 9642.696,E2 9642.696} C_VEL
LIN {X 0,Y 415.027,Z 825.546,A -85,B 0,C 180,E1 9648.154,E2 9648.154} C_VEL
LIN {X 0,Y 417.859,Z 803.812,A -85,B 0,C 180,E1 9653.22,E2 9653.22} C_VEL
LIN {X 0,Y 422.005,Z 777.019,A -85,B 0,C 180,E1 9657.802,E2 9657.802} C_VEL
LIN {X 0,Y 426.933,Z 746.974,A -85,B 0,C 180,E1 9661.672,E2 9661.672} C_VEL
LIN {X 0,Y 432.251,Z 713.132,A -85,B 0,C 180,E1 9664.95,E2 9664.95} C_VEL
LIN {X 0,Y 437.185,Z 676.699,A -85,B 0,C 180,E1 9667.52,E2 9667.52} C_VEL
LIN {X 0,Y 441.524,Z 636.635,A -85,B 0,C 180,E1 9669.414,E2 9669.414} C_VEL
LIN {X 0,Y 442.27,Z 622.022,A -85,B 0,C 180,E1 9669.945,E2 9669.945} C_VEL
LIN {X 0,Y 424.643,Z 582.685,A -85,B 0,C 180,E1 9672.924,E2 9672.924} C_VEL
LIN {X 0,Y 411.317,Z 558.035,A -85,B 0,C 180,E1 9675.135,E2 9675.135} C_VEL
LIN {X 0,Y 411.249,Z 557.03,A -85,B 0,C 180,E1 9675.22,E2 9675.22} C_VEL
LIN {X 0,Y 411.094,Z 557.03,A -85,B 0,C 180,E1 9681.239,E2 9681.239} C_VEL
LIN {X 0,Y 411.17,Z 557.03,A -85,B 0,C 180,E1 9687.88,E2 9687.88} C_VEL
LIN {X 0,Y 411.371,Z 557.03,A -85,B 0,C 180,E1 9693.792,E2 9693.792} C_VEL
LIN {X 0,Y 411.648,Z 557.03,A -85,B 0,C 180,E1 9700.67,E2 9700.67} C_VEL
LIN {X 0,Y 411.699,Z 557.03,A -85,B 0,C 180,E1 9707.253,E2 9707.253} C_VEL
LIN {X 0,Y 412.139,Z 557.03,A -85,B 0,C 180,E1 9713.673,E2 9713.673} C_VEL
LIN {X 0,Y 412.43,Z 557.03,A -85,B 0,C 180,E1 9720,E2 9720} C_VEL
LIN {X 0,Y 412.101,Z 557.03,A -85,B 0,C 180,E1 9726.327,E2 9726.327} C_VEL
LIN {X 0,Y 411.844,Z 557.03,A -85,B 0,C 180,E1 9732.742,E2 9732.742} C_VEL
LIN {X 0,Y 411.656,Z 557.03,A -85,B 0,C 180,E1 9739.329,E2 9739.329} C_VEL
LIN {X 0,Y 411.367,Z 557.03,A -85,B 0,C 180,E1 9746.208,E2 9746.208} C_VEL
LIN {X 0,Y 411.188,Z 557.03,A -85,B 0,C 180,E1 9753.523,E2 9753.523} C_VEL
LIN {X 0,Y 411.032,Z 557.03,A -85,B 0,C 180,E1 9759.326,E2 9759.326} C_VEL
LIN {X 0,Y 411.082,Z 557.03,A -85,B 0,C 180,E1 9765.59,E2 9765.59} C_VEL
LIN {X 0,Y 411.178,Z 557.089,A -85,B 0,C 180,E1 9769.288,E2 9769.288} C_VEL
LIN {X 0,Y 413.655,Z 562.756,A -85,B 0,C 180,E1 9769.73,E2 9769.73} C_VEL
LIN {X 0,Y 435.585,Z 603.8,A -85,B 0,C 180,E1 9773.277,E2 9773.277} C_VEL
LIN {X 0,Y 441.558,Z 617.616,A -85,B 0,C 180,E1 9774.413,E2 9774.413} C_VEL
LIN {X 0,Y 437.834,Z 654.578,A -85,B 0,C 180,E1 9776.085,E2 9776.085} C_VEL
LIN {X 0,Y 432.973,Z 688.605,A -85,B 0,C 180,E1 9778.474,E2 9778.474} C_VEL
LIN {X 0,Y 427.805,Z 718.565,A -85,B 0,C 180,E1 9781.459,E2 9781.459} C_VEL
LIN {X 0,Y 422.657,Z 745.327,A -85,B 0,C 180,E1 9785.107,E2 9785.107} C_VEL
LIN {X 0,Y 418.169,Z 769.066,A -85,B 0,C 180,E1 9789.569,E2 9789.569} C_VEL
LIN {X 0,Y 415.242,Z 786.43,A -85,B 0,C 180,E1 9794.129,E2 9794.129} C_VEL
LIN {X 0,Y 413.545,Z 799.068,A -85,B 0,C 180,E1 9798.918,E2 9798.918} C_VEL
LIN {X 0,Y 412.898,Z 806.861,A -85,B 0,C 180,E1 9803.684,E2 9803.684} C_VEL
LIN {X 0,Y 412.674,Z 810.11,A -85,B 0,C 180,E1 9807.897,E2 9807.897} C_VEL
LIN {X 0,Y 412.724,Z 810.065,A -85,B 0,C 180,E1 9812.102,E2 9812.102} C_VEL
LIN {X 0,Y 413.057,Z 805.367,A -85,B 0,C 180,E1 9817.37,E2 9817.37} C_VEL
LIN {X 0,Y 414.042,Z 795.212,A -85,B 0,C 180,E1 9822.674,E2 9822.674} C_VEL
LIN {X 0,Y 416.135,Z 780.695,A -85,B 0,C 180,E1 9827.467,E2 9827.467} C_VEL
LIN {X 0,Y 419.895,Z 759.842,A -85,B 0,C 180,E1 9832.247,E2 9832.247} C_VEL
LIN {X 0,Y 424.675,Z 734.804,A -85,B 0,C 180,E1 9836.372,E2 9836.372} C_VEL
LIN {X 0,Y 430.078,Z 705.886,A -85,B 0,C 180,E1 9839.833,E2 9839.833} C_VEL
LIN {X 0,Y 435.328,Z 673.392,A -85,B 0,C 180,E1 9842.621,E2 9842.621} C_VEL
LIN {X 0,Y 439.777,Z 638.225,A -85,B 0,C 180,E1 9844.654,E2 9844.654} C_VEL
LIN {X 0,Y 440.912,Z 615.643,A -85,B 0,C 180,E1 9845.634,E2 9845.634} C_VEL
LIN {X 0,Y 423.748,Z 580.577,A -85,B 0,C 180,E1 9848.563,E2 9848.563} C_VEL
LIN {X 0,Y 411.215,Z 558.13,A -85,B 0,C 180,E1 9850.583,E2 9850.583} C_VEL
LIN {X 0,Y 411.122,Z 557.03,A -85,B 0,C 180,E1 9850.779,E2 9850.779} C_VEL
LIN {X 0,Y 411.095,Z 557.03,A -85,B 0,C 180,E1 9857.442,E2 9857.442} C_VEL
LIN {X 0,Y 411.136,Z 557.03,A -85,B 0,C 180,E1 9864.112,E2 9864.112} C_VEL
LIN {X 0,Y 411.331,Z 557.03,A -85,B 0,C 180,E1 9871.414,E2 9871.414} C_VEL
LIN {X 0,Y 411.573,Z 557.03,A -85,B 0,C 180,E1 9878.418,E2 9878.418} C_VEL
LIN {X 0,Y 411.855,Z 557.03,A -85,B 0,C 180,E1 9885.09,E2 9885.09} C_VEL
LIN {X 0,Y 412.055,Z 557.03,A -85,B 0,C 180,E1 9891.549,E2 9891.549} C_VEL
LIN {X 0,Y 412.33,Z 557.03,A -85,B 0,C 180,E1 9897.896,E2 9897.896} C_VEL
LIN {X 0,Y 412.148,Z 557.03,A -85,B 0,C 180,E1 9904.213,E2 9904.213} C_VEL
LIN {X 0,Y 411.875,Z 557.03,A -85,B 0,C 180,E1 9910.591,E2 9910.591} C_VEL
LIN {X 0,Y 411.659,Z 557.03,A -85,B 0,C 180,E1 9917.111,E2 9917.111} C_VEL
LIN {X 0,Y 411.465,Z 557.03,A -85,B 0,C 180,E1 9923.875,E2 9923.875} C_VEL
LIN {X 0,Y 411.328,Z 557.03,A -85,B 0,C 180,E1 9928.587,E2 9928.587} C_VEL
LIN {X 0,Y 411.157,Z 557.03,A -85,B 0,C 180,E1 9936.097,E2 9936.097} C_VEL
LIN {X 0,Y 411.099,Z 557.03,A -85,B 0,C 180,E1 9942.559,E2 9942.559} C_VEL
LIN {X 0,Y 411.319,Z 557.835,A -85,B 0,C 180,E1 9944.869,E2 9944.869} C_VEL
LIN {X 0,Y 434.24,Z 602.464,A -85,B 0,C 180,E1 9948.62,E2 9948.62} C_VEL
LIN {X 0,Y 442.603,Z 624.422,A -85,B 0,C 180,E1 9950.184,E2 9950.184} C_VEL
LIN {X 0,Y 438.831,Z 662.874,A -85,B 0,C 180,E1 9951.727,E2 9951.727} C_VEL
LIN {X 0,Y 434.233,Z 699.179,A -85,B 0,C 180,E1 9953.958,E2 9953.958} C_VEL
LIN {X 0,Y 428.966,Z 734.313,A -85,B 0,C 180,E1 9956.985,E2 9956.985} C_VEL
LIN {X 0,Y 423.732,Z 766.792,A -85,B 0,C 180,E1 9960.764,E2 9960.764} C_VEL
LIN {X 0,Y 419.391,Z 793.857,A -85,B 0,C 180,E1 9964.918,E2 9964.918} C_VEL
LIN {X 0,Y 416.924,Z 810.161,A -85,B 0,C 180,E1 9968.101,E2 9968.101} C_VEL
LIN {X 0,Y 411.823,Z 819.152,A -85,B 0,C 180,E1 9970.065,E2 9970.065} C_VEL
LIN {X 0,Y 406.966,Z 827.151,A -85,B 0,C 180,E1 9972.15,E2 9972.15} C_VEL
LIN {X 0,Y 405.441,Z 841.326,A -85,B 0,C 180,E1 9977.053,E2 9977.053} C_VEL
LIN {X 0,Y 404.848,Z 850.91,A -85,B 0,C 180,E1 9982.169,E2 9982.169} C_VEL
LIN {X 0,Y 404.671,Z 854.715,A -85,B 0,C 180,E1 9985.709,E2 9985.709} C_VEL
LIN {X 0,Y 404.725,Z 856.409,A -85,B 0,C 180,E1 9990,E2 9990} C_VEL
LIN {X 0,Y 404.696,Z 853.813,A -85,B 0,C 180,E1 9995.367,E2 9995.367} C_VEL
LIN {X 0,Y 405.144,Z 845.984,A -85,B 0,C 180,E1 10000.77,E2 10000.77} C_VEL
LIN {X 0,Y 406.366,Z 832.403,A -85,B 0,C 180,E1 10006.227,E2 10006.227} C_VEL
LIN {X 0,Y 408.741,Z 813.278,A -85,B 0,C 180,E1 10011.457,E2 10011.457} C_VEL
LIN {X 0,Y 412.738,Z 788.213,A -85,B 0,C 180,E1 10016.41,E2 10016.41} C_VEL
LIN {X 0,Y 417.954,Z 757.467,A -85,B 0,C 180,E1 10020.911,E2 10020.911} C_VEL
LIN {X 0,Y 423.488,Z 724.985,A -85,B 0,C 180,E1 10024.454,E2 10024.454} C_VEL
LIN {X 0,Y 429.006,Z 688.952,A -85,B 0,C 180,E1 10027.337,E2 10027.337} C_VEL
LIN {X 0,Y 433.737,Z 651.652,A -85,B 0,C 180,E1 10029.41,E2 10029.41} C_VEL
LIN {X 0,Y 435.76,Z 624.588,A -85,B 0,C 180,E1 10030.493,E2 10030.493} C_VEL
LIN {X 0,Y 419.916,Z 588.391,A -85,B 0,C 180,E1 10033.342,E2 10033.342} C_VEL
LIN {X 0,Y 403.285,Z 557.848,A -85,B 0,C 180,E1 10036.204,E2 10036.204} C_VEL
LIN {X 0,Y 403.193,Z 557.03,A -85,B 0,C 180,E1 10037.477,E2 10037.477} C_VEL
LIN {X 0,Y 403.144,Z 557.03,A -85,B 0,C 180,E1 10043.068,E2 10043.068} C_VEL
LIN {X 0,Y 403.269,Z 557.03,A -85,B 0,C 180,E1 10049.715,E2 10049.715} C_VEL
LIN {X 0,Y 403.49,Z 557.03,A -85,B 0,C 180,E1 10055.623,E2 10055.623} C_VEL
LIN {X 0,Y 403.717,Z 557.03,A -85,B 0,C 180,E1 10062.542,E2 10062.542} C_VEL
LIN {X 0,Y 403.855,Z 557.03,A -85,B 0,C 180,E1 10069.196,E2 10069.196} C_VEL
LIN {X 0,Y 404.241,Z 557.03,A -85,B 0,C 180,E1 10075.704,E2 10075.704} C_VEL
LIN {X 0,Y 404.452,Z 557.03,A -85,B 0,C 180,E1 10082.145,E2 10082.145} C_VEL
LIN {X 0,Y 404.114,Z 557.03,A -85,B 0,C 180,E1 10088.618,E2 10088.618} C_VEL
LIN {X 0,Y 403.841,Z 557.03,A -85,B 0,C 180,E1 10095.213,E2 10095.213} C_VEL
LIN {X 0,Y 403.611,Z 557.03,A -85,B 0,C 180,E1 10102.03,E2 10102.03} C_VEL
LIN {X 0,Y 403.329,Z 557.03,A -85,B 0,C 180,E1 10109.207,E2 10109.207} C_VEL
LIN {X 0,Y 403.21,Z 557.03,A -85,B 0,C 180,E1 10114.299,E2 10114.299} C_VEL
LIN {X 0,Y 403.094,Z 557.03,A -85,B 0,C 180,E1 10121.304,E2 10121.304} C_VEL
LIN {X 0,Y 403.176,Z 557.03,A -85,B 0,C 180,E1 10128.195,E2 10128.195} C_VEL
LIN {X 0,Y 405.854,Z 562.929,A -85,B 0,C 180,E1 10128.713,E2 10128.713} C_VEL
LIN {X 0,Y 427.033,Z 601.728,A -85,B 0,C 180,E1 10132.268,E2 10132.268} C_VEL
LIN {X 0,Y 435.107,Z 620.671,A -85,B 0,C 180,E1 10133.879,E2 10133.879} C_VEL
LIN {X 0,Y 431.198,Z 656.622,A -85,B 0,C 180,E1 10135.572,E2 10135.572} C_VEL
LIN {X 0,Y 426.111,Z 690.345,A -85,B 0,C 180,E1 10138.007,E2 10138.007} C_VEL
LIN {X 0,Y 420.449,Z 721.441,A -85,B 0,C 180,E1 10141.207,E2 10141.207} C_VEL
LIN {X 0,Y 414.758,Z 749.13,A -85,B 0,C 180,E1 10145.178,E2 10145.178} C_VEL
LIN {X 0,Y 410.416,Z 770.892,A -85,B 0,C 180,E1 10149.484,E2 10149.484} C_VEL
LIN {X 0,Y 407.31,Z 788.582,A -85,B 0,C 180,E1 10154.365,E2 10154.365} C_VEL
LIN {X 0,Y 405.582,Z 801.708,A -85,B 0,C 180,E1 10159.786,E2 10159.786} C_VEL
LIN {X 0,Y 404.978,Z 808.451,A -85,B 0,C 180,E1 10164.637,E2 10164.637} C_VEL
LIN {X 0,Y 404.842,Z 810.978,A -85,B 0,C 180,E1 10170,E2 10170} C_VEL
LIN {X 0,Y 405,Z 808.35,A -85,B 0,C 180,E1 10175.362,E2 10175.362} C_VEL
LIN {X 0,Y 405.696,Z 800.445,A -85,B 0,C 180,E1 10180.754,E2 10180.754} C_VEL
LIN {X 0,Y 407.389,Z 788.305,A -85,B 0,C 180,E1 10185.631,E2 10185.631} C_VEL
LIN {X 0,Y 410.726,Z 769.37,A -85,B 0,C 180,E1 10190.781,E2 10190.781} C_VEL
LIN {X 0,Y 415.548,Z 745.37,A -85,B 0,C 180,E1 10195.347,E2 10195.347} C_VEL
LIN {X 0,Y 421.149,Z 717.38,A -85,B 0,C 180,E1 10199.181,E2 10199.181} C_VEL
LIN {X 0,Y 426.925,Z 685.759,A -85,B 0,C 180,E1 10202.288,E2 10202.288} C_VEL
LIN {X 0,Y 431.945,Z 651.277,A -85,B 0,C 180,E1 10204.637,E2 10204.637} C_VEL
LIN {X 0,Y 434.585,Z 618.602,A -85,B 0,C 180,E1 10206.177,E2 10206.177} C_VEL
LIN {X 0,Y 417.327,Z 582.886,A -85,B 0,C 180,E1 10209.283,E2 10209.283} C_VEL
LIN {X 0,Y 403.212,Z 558.056,A -85,B 0,C 180,E1 10211.653,E2 10211.653} C_VEL
LIN {X 0,Y 403.159,Z 557.03,A -85,B 0,C 180,E1 10211.967,E2 10211.967} C_VEL
